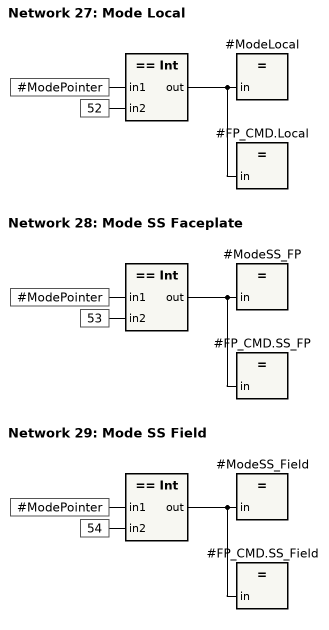
   #ModeLocal := #ModePointer = 52;
   #FP_CMD.Local := #ModeLocal;
END_REGION

REGION Network 28: Mode SS Faceplate
   #ModeSS_FP := #ModePointer = 53;
   #FP_CMD.SS_FP := #ModeSS_FP;
END_REGION

REGION Network 29: Mode SS Field
   #ModeSS_Field := #ModePointer = 54;
   #FP_CMD.SS_Field := #ModeSS_Field;
END_REGION

REGION Network 30: FACEPLATE COMMANDS (Pulse Type)
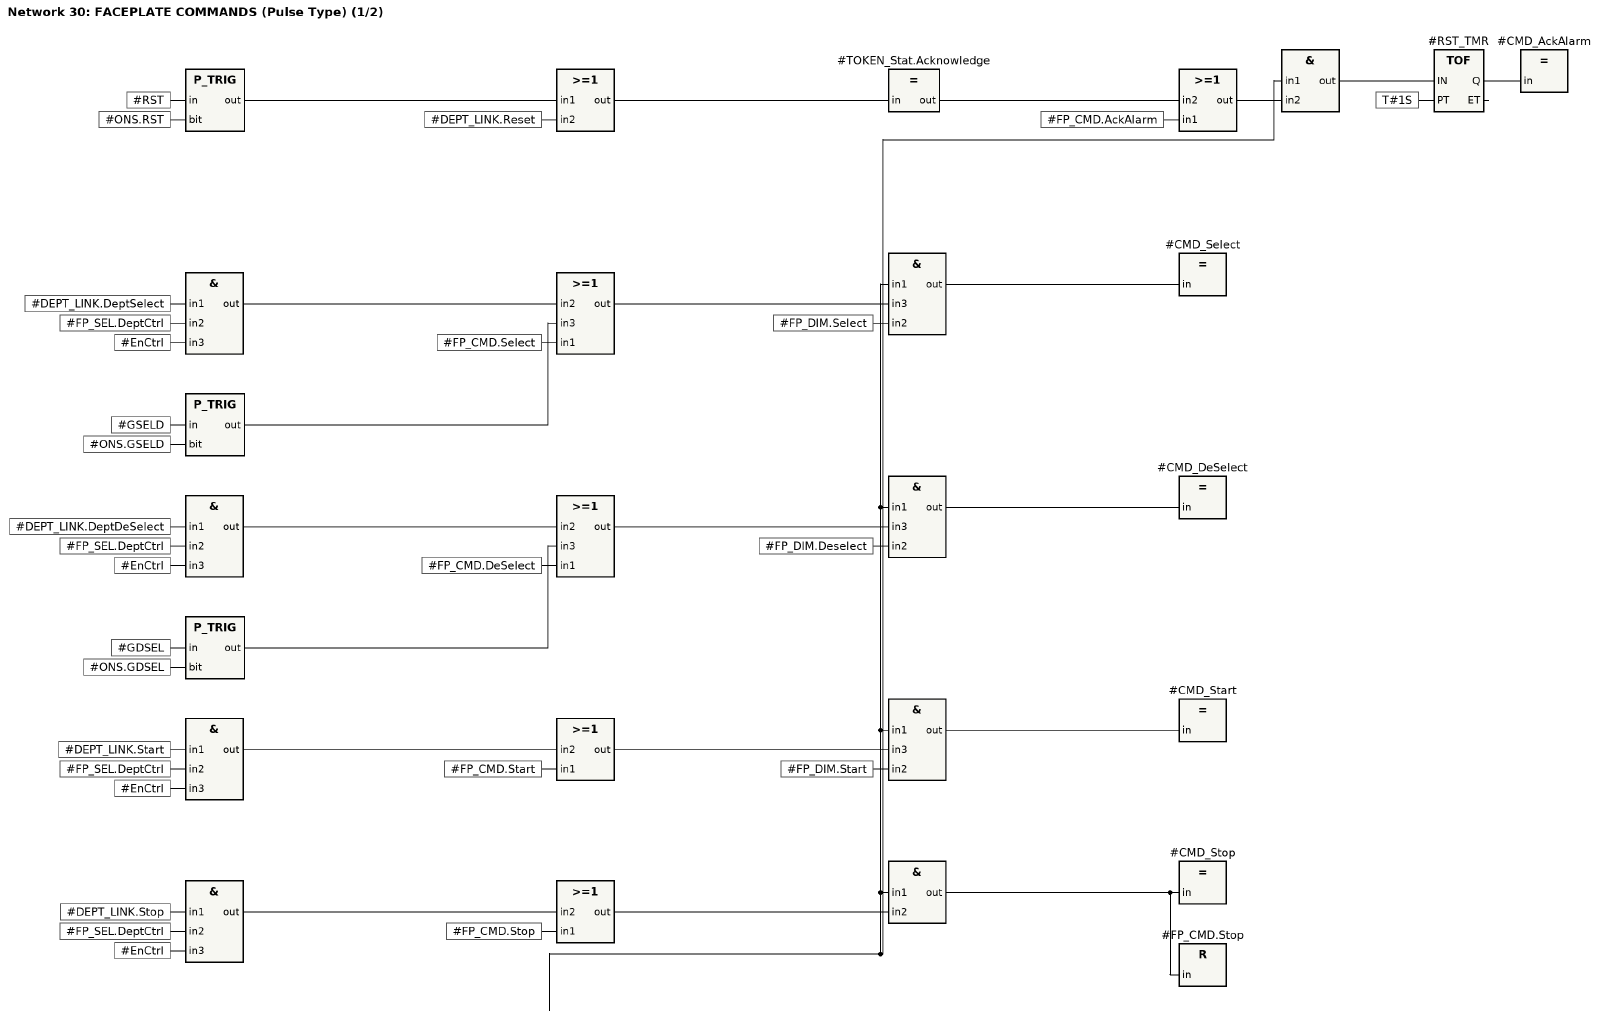
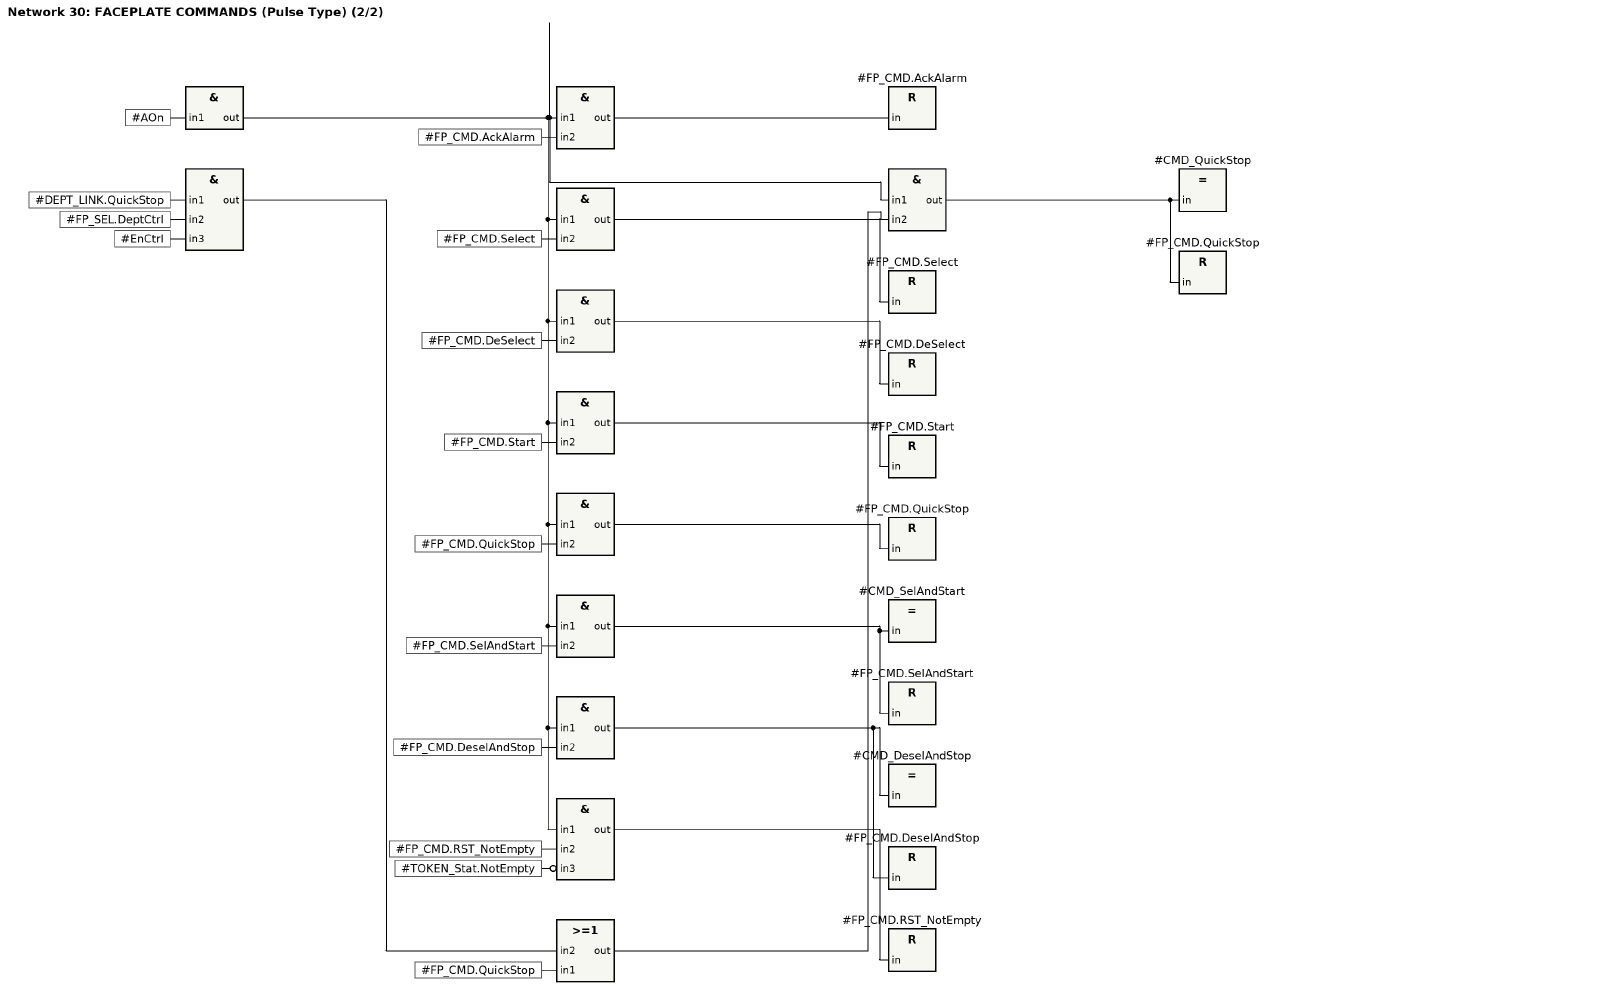
   #_w1 := #RST AND NOT #ONS.RST;   // rising edge
   #ONS.RST := #RST;
   #TOKEN_Stat.Acknowledge := #_w1 OR #DEPT_LINK.Reset;
   #RST_TMR(IN := #AOn AND (#TOKEN_Stat.Acknowledge OR #FP_CMD.AckAlarm), PT := T#1S);   // TOF
   #CMD_AckAlarm := #RST_TMR.Q;
   IF #AOn AND #FP_CMD.AckAlarm THEN #FP_CMD.AckAlarm := FALSE; END_IF;
   #_w2 := #GSELD AND NOT #ONS.GSELD;   // rising edge
   #ONS.GSELD := #GSELD;
   #CMD_Select := #AOn AND ((#DEPT_LINK.DeptSelect AND #FP_SEL.DeptCtrl AND #EnCtrl) OR #_w2 OR #FP_CMD.Select) AND #FP_DIM.Select;
   IF #AOn AND #FP_CMD.Select THEN #FP_CMD.Select := FALSE; END_IF;
   #_w3 := #GDSEL AND NOT #ONS.GDSEL;   // rising edge
   #ONS.GDSEL := #GDSEL;
   #CMD_DeSelect := #AOn AND ((#DEPT_LINK.DeptDeSelect AND #FP_SEL.DeptCtrl AND #EnCtrl) OR #_w3 OR #FP_CMD.DeSelect) AND #FP_DIM.Deselect;
   IF #AOn AND #FP_CMD.DeSelect THEN #FP_CMD.DeSelect := FALSE; END_IF;
   #CMD_Start := #AOn AND ((#DEPT_LINK.Start AND #FP_SEL.DeptCtrl AND #EnCtrl) OR #FP_CMD.Start) AND #FP_DIM.Start;
   IF #AOn AND #FP_CMD.Start THEN #FP_CMD.Start := FALSE; END_IF;
   #CMD_Stop := #AOn AND ((#DEPT_LINK.Stop AND #FP_SEL.DeptCtrl AND #EnCtrl) OR #FP_CMD.Stop);
   IF #CMD_Stop THEN #FP_CMD.Stop := FALSE; END_IF;
   #CMD_QuickStop := #AOn AND ((#DEPT_LINK.QuickStop AND #FP_SEL.DeptCtrl AND #EnCtrl) OR #FP_CMD.QuickStop);
   IF #CMD_QuickStop THEN #FP_CMD.QuickStop := FALSE; END_IF;
   IF #AOn AND #FP_CMD.QuickStop THEN #FP_CMD.QuickStop := FALSE; END_IF;
   #CMD_SelAndStart := #AOn AND #FP_CMD.SelAndStart;
   IF #CMD_SelAndStart THEN #FP_CMD.SelAndStart := FALSE; END_IF;
   #CMD_DeselAndStop := #AOn AND #FP_CMD.DeselAndStop;
   IF #CMD_DeselAndStop THEN #FP_CMD.DeselAndStop := FALSE; END_IF;
   IF #AOn AND #FP_CMD.RST_NotEmpty AND NOT #TOKEN_Stat.NotEmpty THEN #FP_CMD.RST_NotEmpty := FALSE; END_IF;
END_REGION

REGION Network 31: Start Warning timer
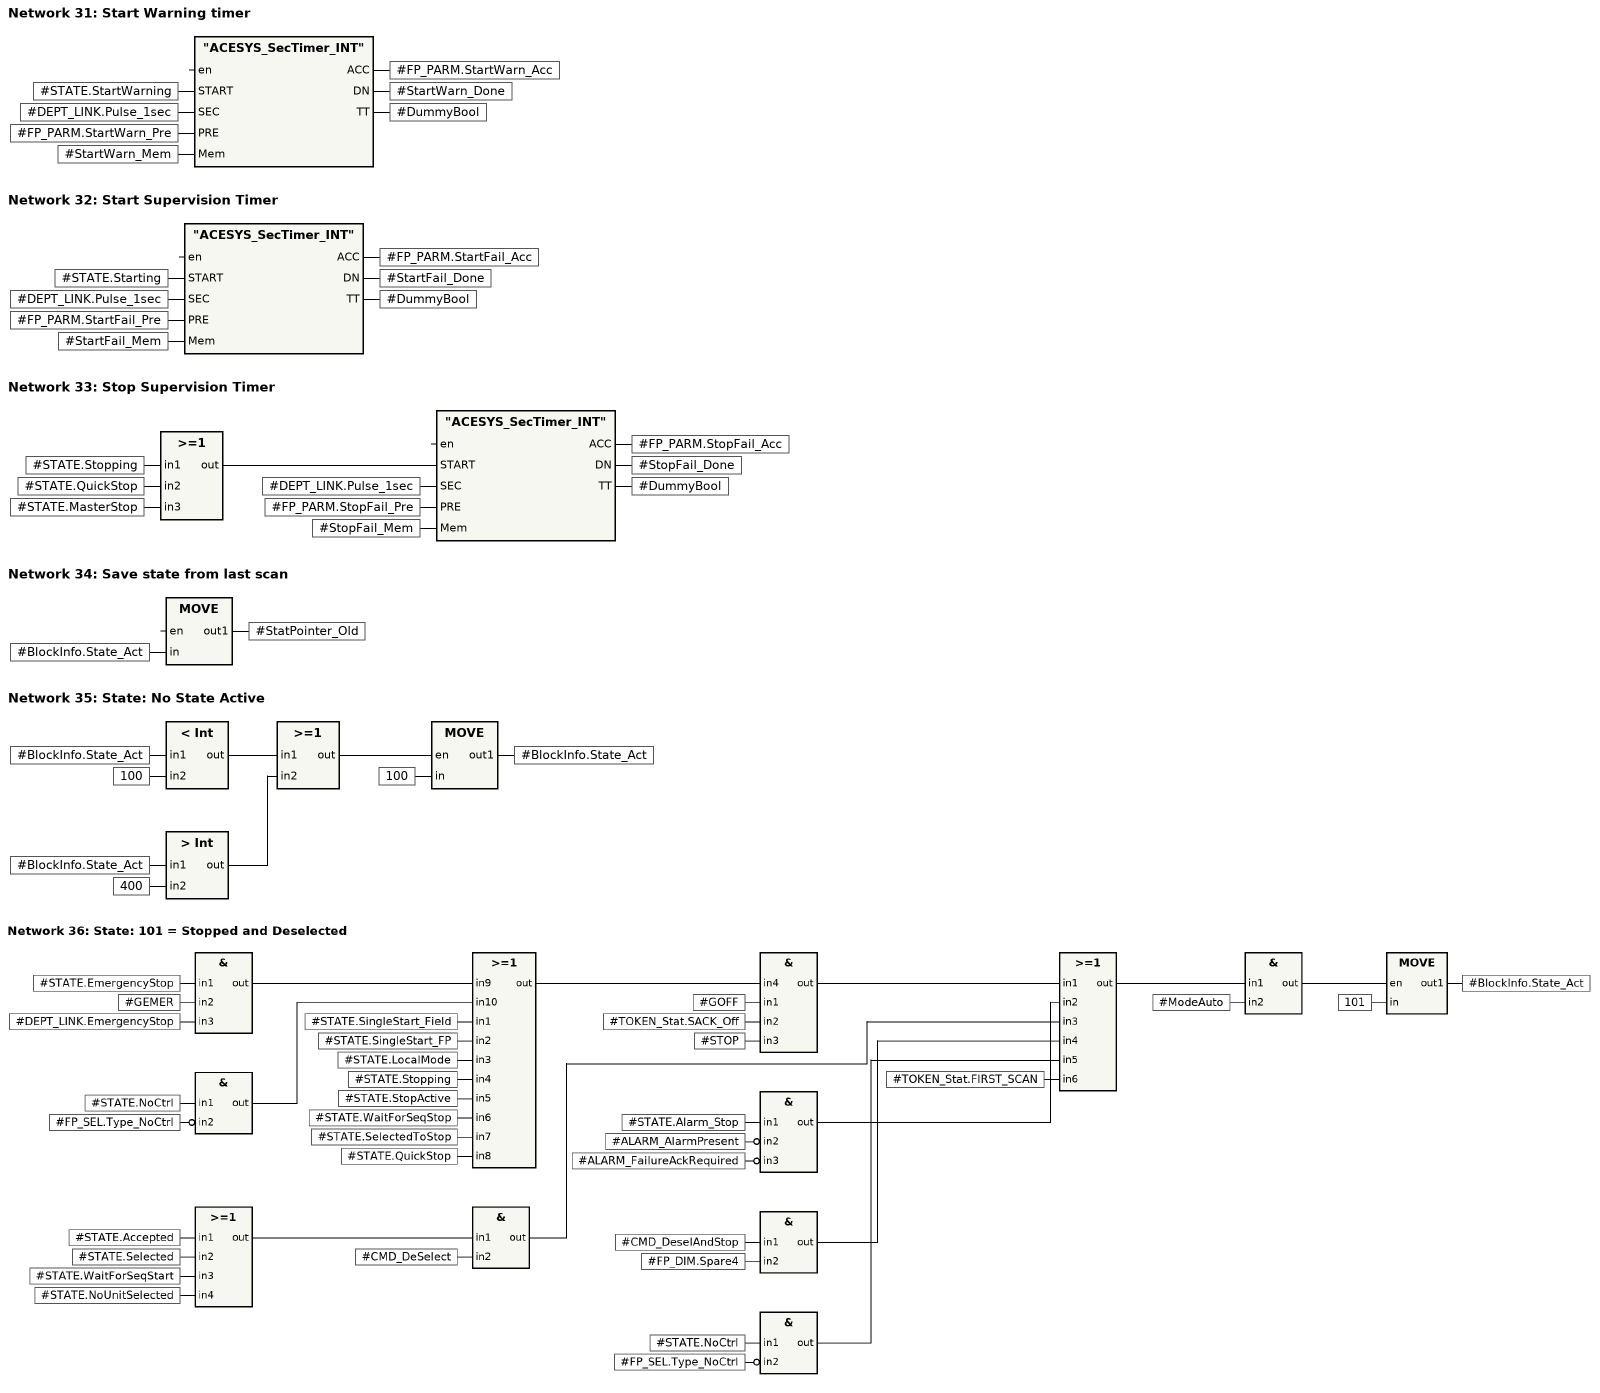
   "ACESYS_SecTimer_INT"(START := #STATE.StartWarning,
                         SEC := #DEPT_LINK.Pulse_1sec,
                         PRE := #FP_PARM.StartWarn_Pre,
                         Mem := #StartWarn_Mem,
                         ACC => #FP_PARM.StartWarn_Acc,
                         DN => #StartWarn_Done,
                         TT => #DummyBool);
END_REGION

REGION Network 32: Start Supervision Timer
   "ACESYS_SecTimer_INT"(START := #STATE.Starting,
                         SEC := #DEPT_LINK.Pulse_1sec,
                         PRE := #FP_PARM.StartFail_Pre,
                         Mem := #StartFail_Mem,
                         ACC => #FP_PARM.StartFail_Acc,
                         DN => #StartFail_Done,
                         TT => #DummyBool);
END_REGION

REGION Network 33: Stop Supervision Timer
   "ACESYS_SecTimer_INT"(START := #STATE.Stopping OR #STATE.QuickStop OR #STATE.MasterStop,
                         SEC := #DEPT_LINK.Pulse_1sec,
                         PRE := #FP_PARM.StopFail_Pre,
                         Mem := #StopFail_Mem,
                         ACC => #FP_PARM.StopFail_Acc,
                         DN => #StopFail_Done,
                         TT => #DummyBool);
END_REGION

REGION Network 34: Save state from last scan
   #StatPointer_Old := #BlockInfo.State_Act;
END_REGION

REGION Network 35: State: No State Active
   IF (#BlockInfo.State_Act < 100) OR (#BlockInfo.State_Act > 400) THEN #BlockInfo.State_Act := 100; END_IF;
END_REGION

REGION Network 36: State: 101 = Stopped and Deselected
   // Build 004 - 05.Aug.2021 (MIA-US): Transition from State_WaitForSeqStop added
   IF ((((#STATE.EmergencyStop AND #GEMER AND #DEPT_LINK.EmergencyStop) OR (#STATE.NoCtrl AND NOT #FP_SEL.Type_NoCtrl) OR #STATE.SingleStart_Field OR #STATE.SingleStart_FP OR #STATE.LocalMode OR #STATE.Stopping OR #STATE.StopActive OR #STATE.WaitForSeqStop OR #STATE.SelectedToStop OR #STATE.QuickStop) AND #GOFF AND #TOKEN_Stat.SACK_Off AND #STOP) OR (#STATE.Alarm_Stop AND NOT #ALARM_AlarmPresent AND NOT #ALARM_FailureAckRequired) OR ((#STATE.Accepted OR #STATE.Selected OR #STATE.WaitForSeqStart OR #STATE.NoUnitSelected) AND #CMD_DeSelect) OR (#CMD_DeselAndStop AND #FP_DIM.Spare4) OR (#STATE.NoCtrl AND NOT #FP_SEL.Type_NoCtrl) OR #TOKEN_Stat.FIRST_SCAN) AND #ModeAuto THEN
       #BlockInfo.State_Act := 101;
   END_IF;
END_REGION

REGION Network 37 (SCL): Transfer Interlock OK to Stat
   #OUT.INTL_OK_STAT := PEEK_BOOL(area :=16#84, dbNumber := #BlockInfo.DB_Number, byteOffset := 2, bitOffset := 0);
   #OUT.INTL_SEQ_STR_OK_STAT := PEEK_BOOL(area := 16#84, dbNumber := #BlockInfo.DB_Number, byteOffset := 4, bitOffset := 0);
   #OUT.INTL_SEQ_STP_OK_STAT := PEEK_BOOL(area := 16#84, dbNumber := #BlockInfo.DB_Number, byteOffset := 6, bitOffset := 0);
END_REGION

REGION Network 38: Conditions for Accept
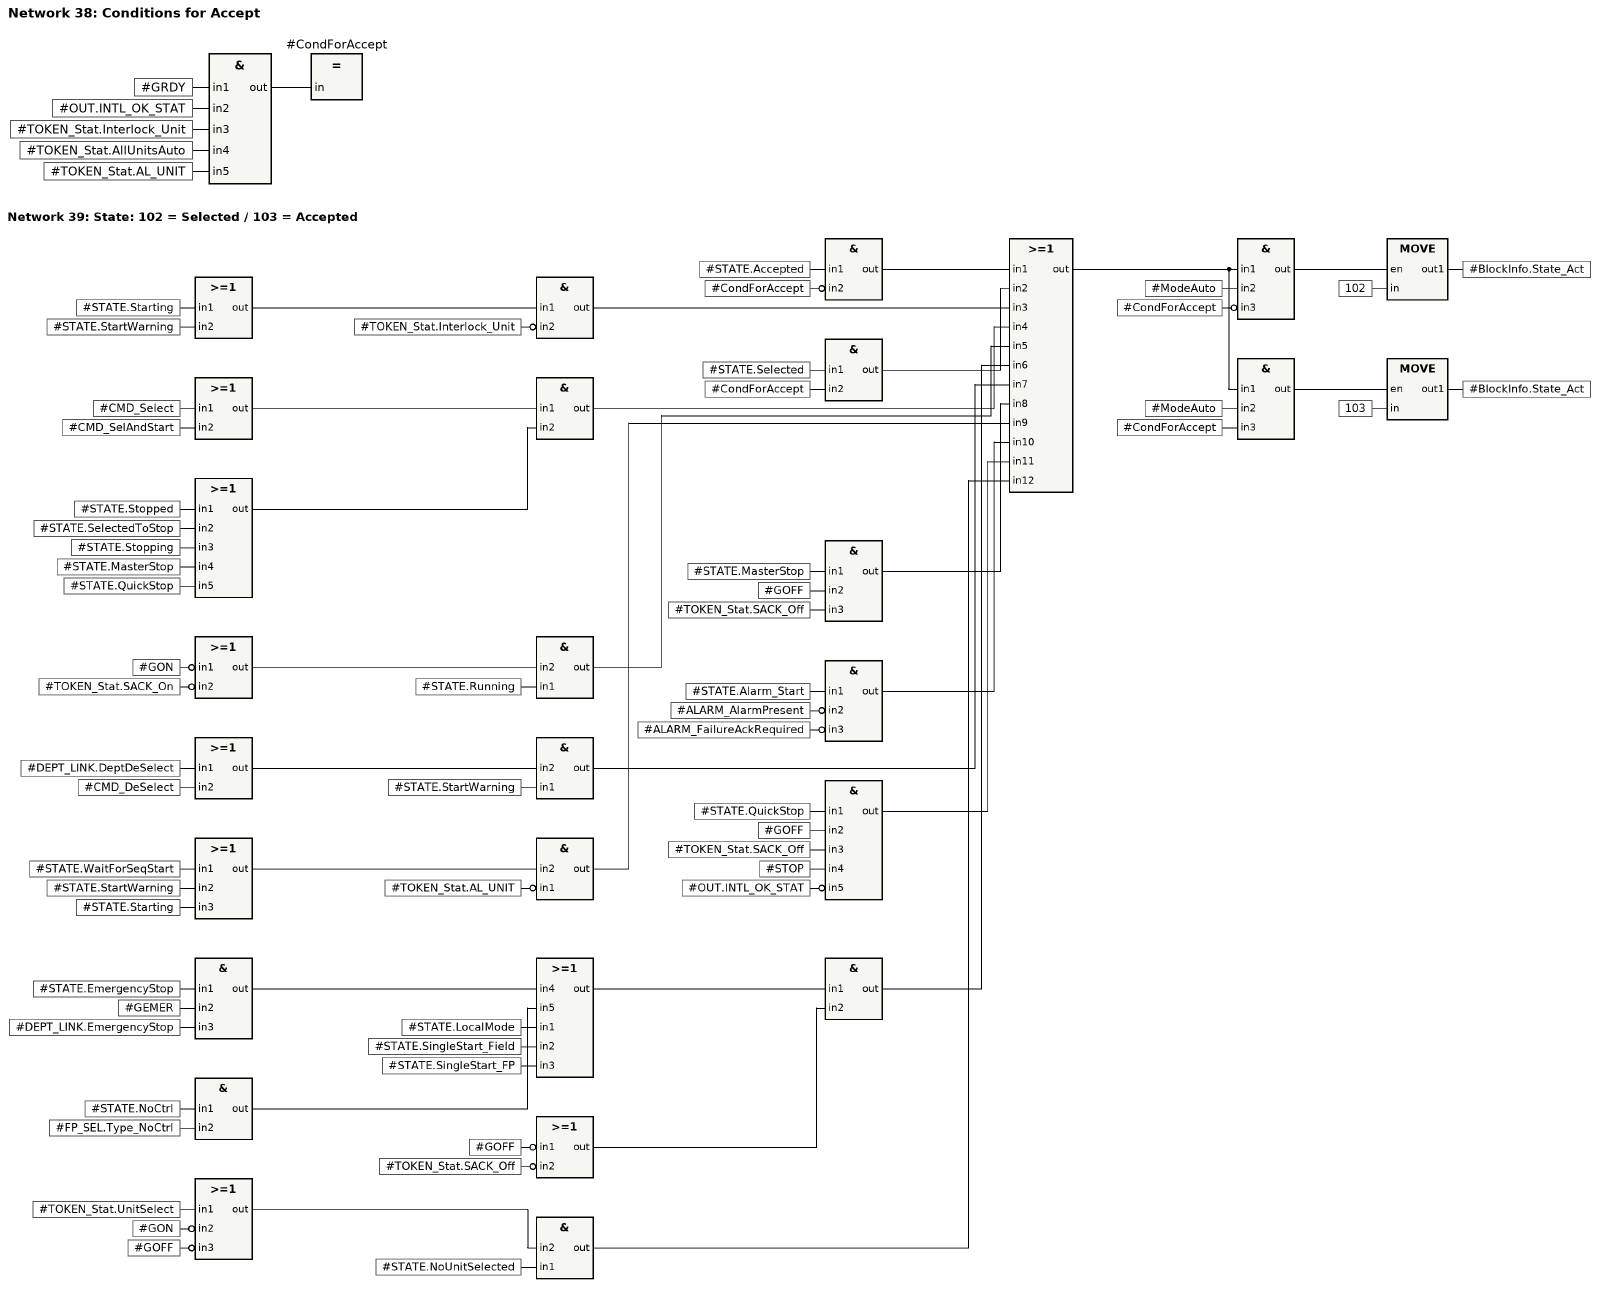
   #CondForAccept := #GRDY AND #OUT.INTL_OK_STAT AND #TOKEN_Stat.Interlock_Unit AND #TOKEN_Stat.AllUnitsAuto AND #TOKEN_Stat.AL_UNIT;
END_REGION

REGION Network 39: State: 102 = Selected / 103 = Accepted
   #_w1 := (#STATE.Accepted AND NOT #CondForAccept) OR (#STATE.Selected AND #CondForAccept) OR ((#STATE.Starting OR #STATE.StartWarning) AND NOT #TOKEN_Stat.Interlock_Unit) OR ((#CMD_Select OR #CMD_SelAndStart) AND (#STATE.Stopped OR #STATE.SelectedToStop OR #STATE.Stopping OR #STATE.MasterStop OR #STATE.QuickStop)) OR ((NOT #GON OR NOT #TOKEN_Stat.SACK_On) AND #STATE.Running) OR (((#STATE.EmergencyStop AND #GEMER AND #DEPT_LINK.EmergencyStop) OR (#STATE.NoCtrl AND #FP_SEL.Type_NoCtrl) OR #STATE.LocalMode OR #STATE.SingleStart_Field OR #STATE.SingleStart_FP) AND (NOT #GOFF OR NOT #TOKEN_Stat.SACK_Off)) OR ((#DEPT_LINK.DeptDeSelect OR #CMD_DeSelect) AND #STATE.StartWarning) OR (#STATE.MasterStop AND #GOFF AND #TOKEN_Stat.SACK_Off) OR ((#STATE.WaitForSeqStart OR #STATE.StartWarning OR #STATE.Starting) AND NOT #TOKEN_Stat.AL_UNIT) OR (#STATE.Alarm_Start AND NOT #ALARM_AlarmPresent AND NOT #ALARM_FailureAckRequired) OR (#STATE.QuickStop AND #GOFF AND #TOKEN_Stat.SACK_Off AND #STOP AND NOT #OUT.INTL_OK_STAT) OR ((#TOKEN_Stat.UnitSelect OR NOT #GON OR NOT #GOFF) AND #STATE.NoUnitSelected);
   IF #_w1 AND #ModeAuto AND NOT #CondForAccept THEN #BlockInfo.State_Act := 102; END_IF;
   IF #_w1 AND #ModeAuto AND #CondForAccept THEN #BlockInfo.State_Act := 103; END_IF;
END_REGION

REGION Network 40: State: 104 = Wait for Sequence Start
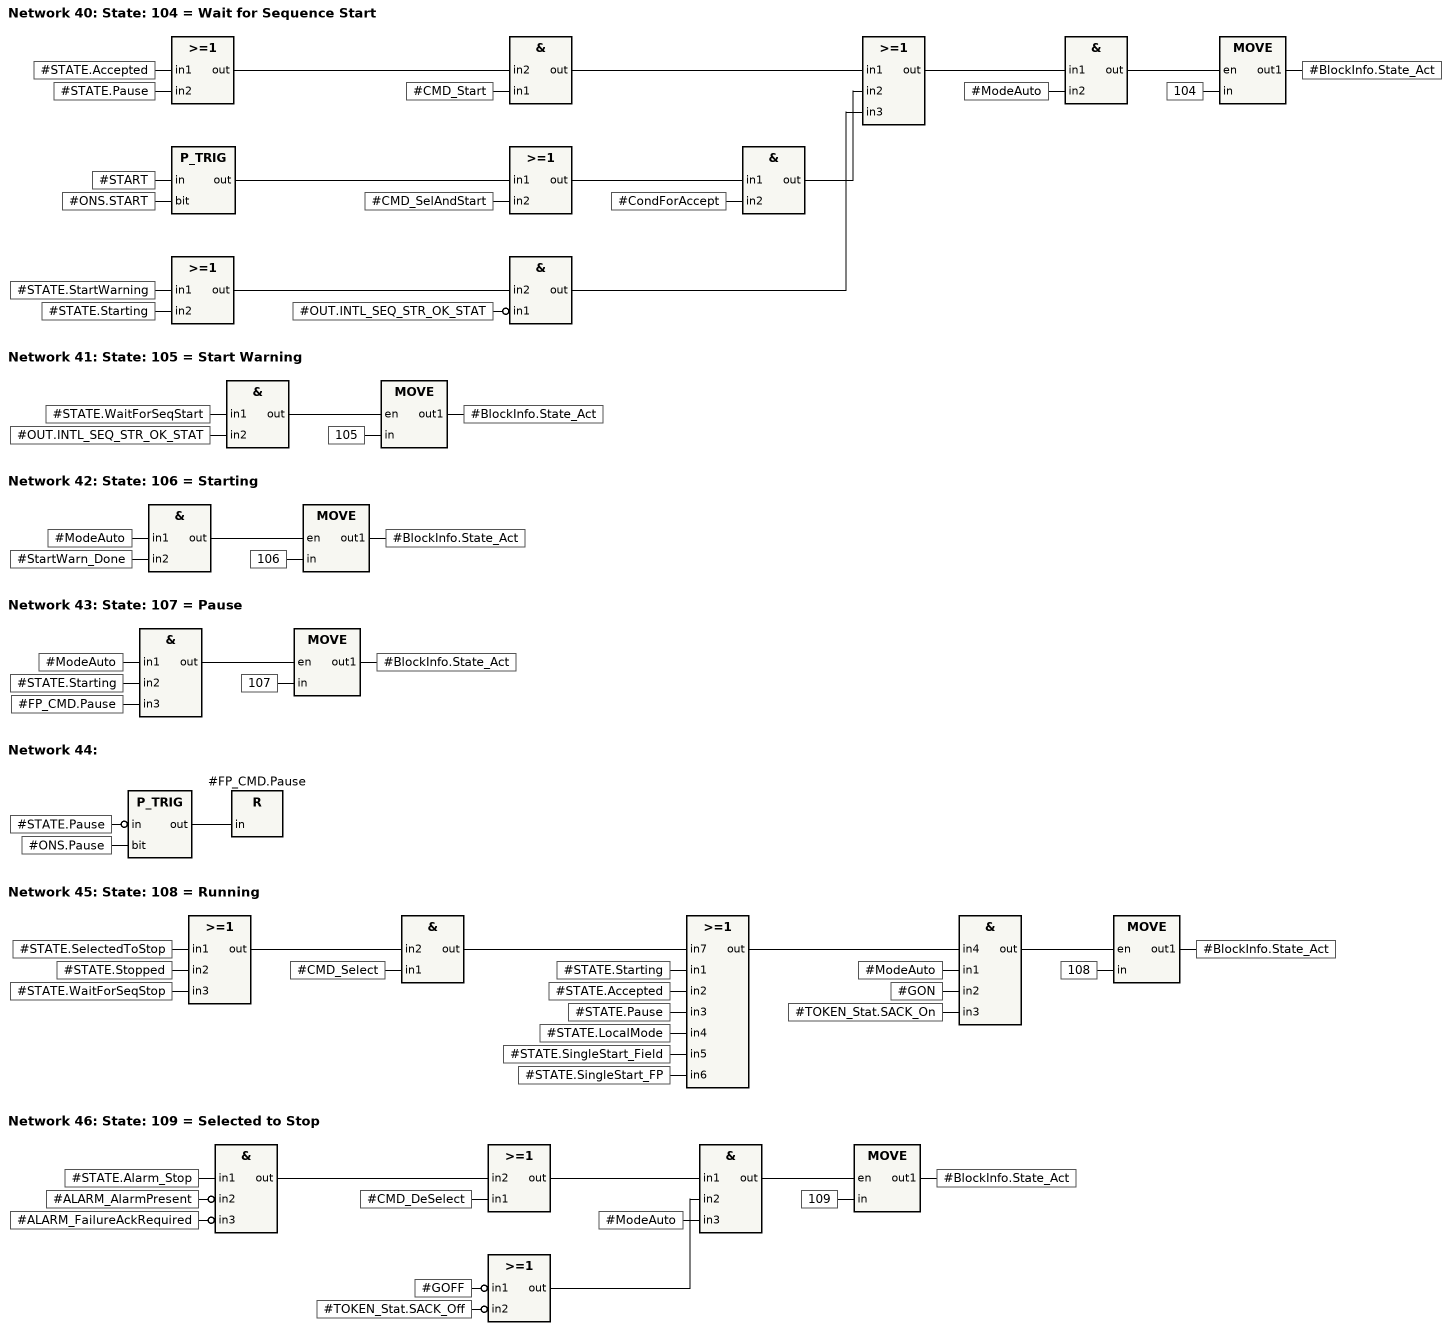
   #_w1 := #START AND NOT #ONS.START;   // rising edge
   #ONS.START := #START;
   IF (((#STATE.Accepted OR #STATE.Pause) AND #CMD_Start) OR ((#_w1 OR #CMD_SelAndStart) AND #CondForAccept) OR ((#STATE.StartWarning OR #STATE.Starting) AND NOT #OUT.INTL_SEQ_STR_OK_STAT)) AND #ModeAuto THEN
       #BlockInfo.State_Act := 104;
   END_IF;
END_REGION

REGION Network 41: State: 105 = Start Warning
   IF #STATE.WaitForSeqStart AND #OUT.INTL_SEQ_STR_OK_STAT THEN #BlockInfo.State_Act := 105; END_IF;
END_REGION

REGION Network 42: State: 106 = Starting
   IF #ModeAuto AND #StartWarn_Done THEN #BlockInfo.State_Act := 106; END_IF;
END_REGION

REGION Network 43: State: 107 = Pause
   IF #ModeAuto AND #STATE.Starting AND #FP_CMD.Pause THEN #BlockInfo.State_Act := 107; END_IF;
END_REGION

REGION Network 44
   #_w1 := NOT #STATE.Pause AND NOT #ONS.Pause;   // rising edge
   #ONS.Pause := NOT #STATE.Pause;
   IF #_w1 THEN #FP_CMD.Pause := FALSE; END_IF;
END_REGION

REGION Network 45: State: 108 = Running
   IF (((#STATE.SelectedToStop OR #STATE.Stopped OR #STATE.WaitForSeqStop) AND #CMD_Select) OR #STATE.Starting OR #STATE.Accepted OR #STATE.Pause OR #STATE.LocalMode OR #STATE.SingleStart_Field OR #STATE.SingleStart_FP) AND #ModeAuto AND #GON AND #TOKEN_Stat.SACK_On THEN
       #BlockInfo.State_Act := 108;
   END_IF;
END_REGION

REGION Network 46: State: 109 = Selected to Stop
   IF ((#STATE.Alarm_Stop AND NOT #ALARM_AlarmPresent AND NOT #ALARM_FailureAckRequired) OR #CMD_DeSelect) AND (NOT #GOFF OR NOT #TOKEN_Stat.SACK_Off) AND #ModeAuto THEN
       #BlockInfo.State_Act := 109;
   END_IF;
END_REGION

REGION Network 47: State: 110 = Wait for Sequence Stop
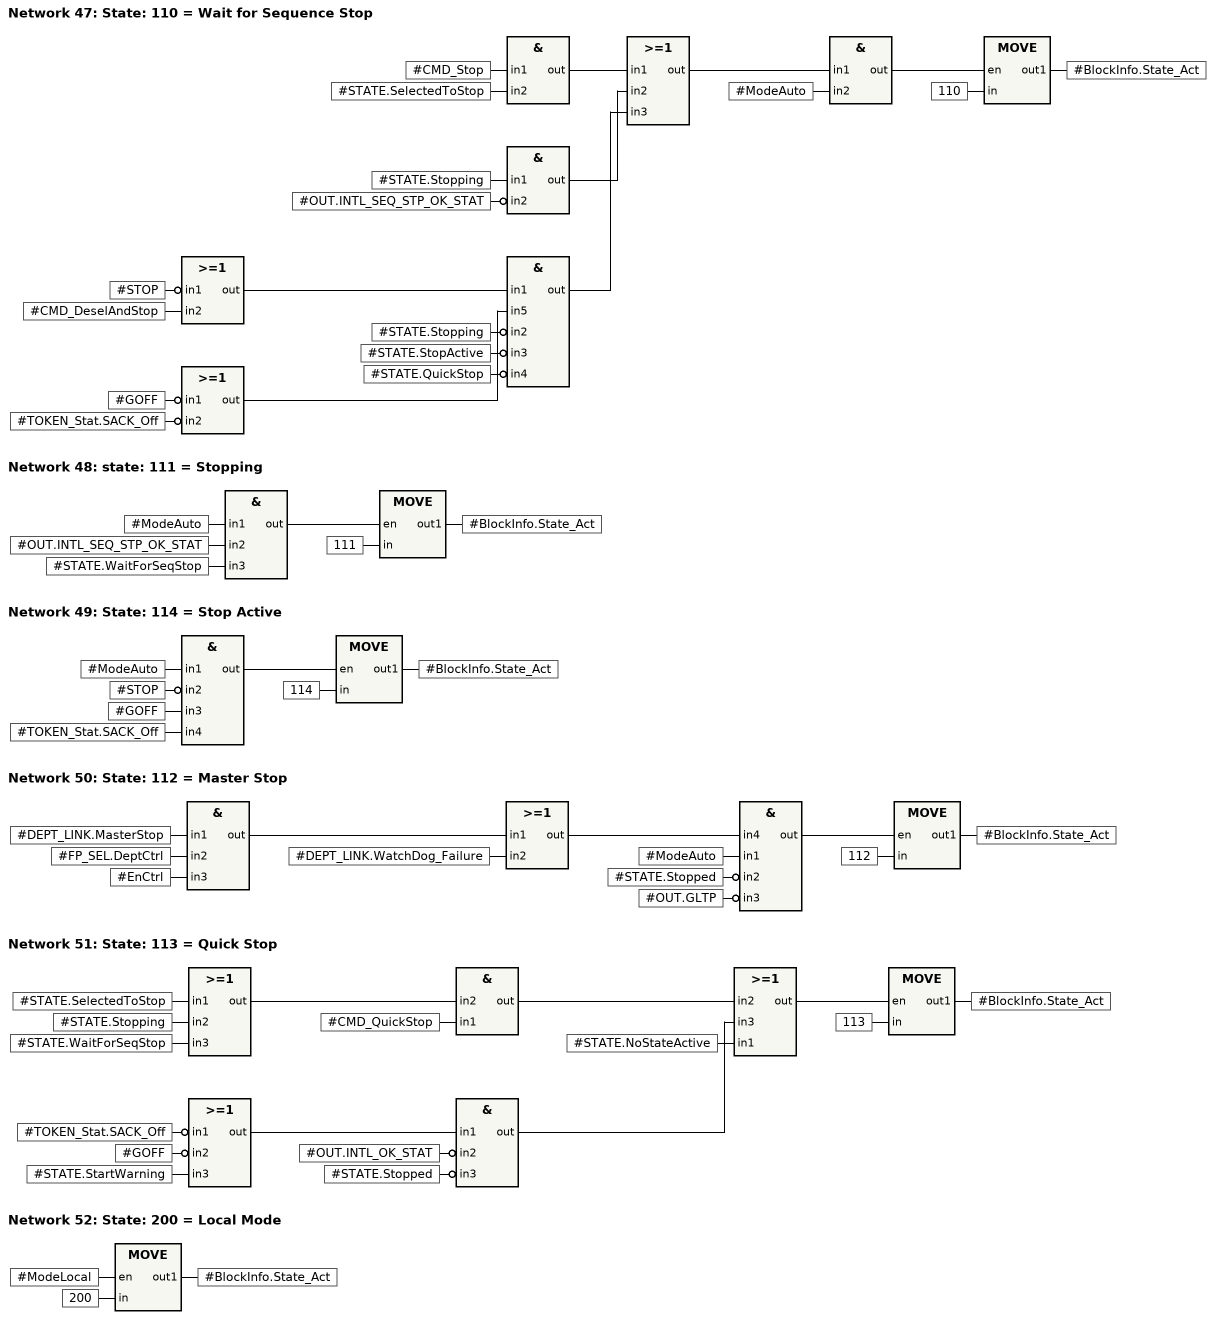
   IF ((#CMD_Stop AND #STATE.SelectedToStop) OR (#STATE.Stopping AND NOT #OUT.INTL_SEQ_STP_OK_STAT) OR ((NOT #STOP OR #CMD_DeselAndStop) AND (NOT #GOFF OR NOT #TOKEN_Stat.SACK_Off) AND NOT #STATE.Stopping AND NOT #STATE.StopActive AND NOT #STATE.QuickStop)) AND #ModeAuto THEN
       #BlockInfo.State_Act := 110;
   END_IF;
END_REGION

REGION Network 48: state: 111 = Stopping
   IF #ModeAuto AND #OUT.INTL_SEQ_STP_OK_STAT AND #STATE.WaitForSeqStop THEN
       #BlockInfo.State_Act := 111;
   END_IF;
END_REGION

REGION Network 49: State: 114 = Stop Active
   IF #ModeAuto AND NOT #STOP AND #GOFF AND #TOKEN_Stat.SACK_Off THEN #BlockInfo.State_Act := 114; END_IF;
END_REGION

REGION Network 50: State: 112 = Master Stop
   IF ((#DEPT_LINK.MasterStop AND #FP_SEL.DeptCtrl AND #EnCtrl) OR #DEPT_LINK.WatchDog_Failure) AND #ModeAuto AND NOT #STATE.Stopped AND NOT #OUT.GLTP THEN
       #BlockInfo.State_Act := 112;
   END_IF;
END_REGION

REGION Network 51: State: 113 = Quick Stop
   // Build 002 - 17.Dec.2019 (MIA-US): Added STATE.StartWarning to allow transition to "Interlock" state when INTL=0 during start warning
   // Build 003 - 24.Jun.2020 (MIA-US): Removed TOKEN_Stat.SACK_On
   IF ((#STATE.SelectedToStop OR #STATE.Stopping OR #STATE.WaitForSeqStop) AND #CMD_QuickStop) OR ((NOT #TOKEN_Stat.SACK_Off OR NOT #GOFF OR #STATE.StartWarning) AND NOT #OUT.INTL_OK_STAT AND NOT #STATE.Stopped) OR #STATE.NoStateActive THEN
       #BlockInfo.State_Act := 113;
   END_IF;
END_REGION

REGION Network 52: State: 200 = Local Mode
   IF #ModeLocal THEN #BlockInfo.State_Act := 200; END_IF;
END_REGION

REGION Network 53: State: 250 = Single Start from Faceplate
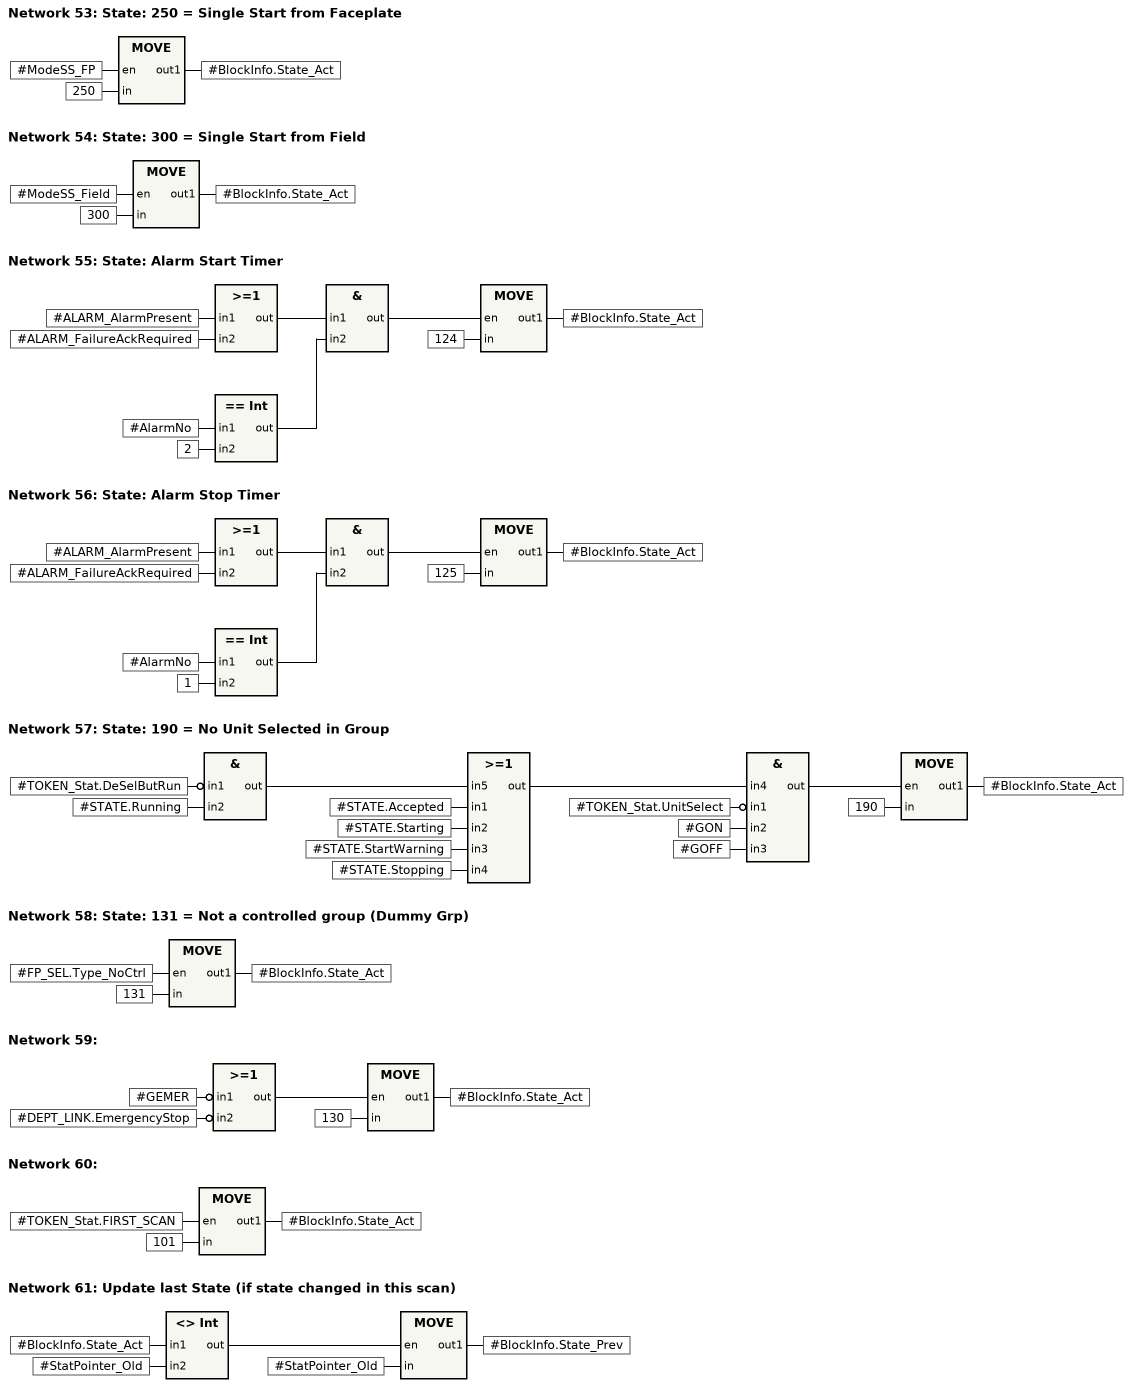
   IF #ModeSS_FP THEN #BlockInfo.State_Act := 250; END_IF;
END_REGION

REGION Network 54: State: 300 = Single Start from Field
   IF #ModeSS_Field THEN #BlockInfo.State_Act := 300; END_IF;
END_REGION

REGION Network 55: State: Alarm Start Timer
   IF (#ALARM_AlarmPresent OR #ALARM_FailureAckRequired) AND (#AlarmNo = 2) THEN
       #BlockInfo.State_Act := 124;
   END_IF;
END_REGION

REGION Network 56: State: Alarm Stop Timer
   IF (#ALARM_AlarmPresent OR #ALARM_FailureAckRequired) AND (#AlarmNo = 1) THEN
       #BlockInfo.State_Act := 125;
   END_IF;
END_REGION

REGION Network 57: State: 190 = No Unit Selected in Group
   IF ((NOT #TOKEN_Stat.DeSelButRun AND #STATE.Running) OR #STATE.Accepted OR #STATE.Starting OR #STATE.StartWarning OR #STATE.Stopping) AND NOT #TOKEN_Stat.UnitSelect AND #GON AND #GOFF THEN
       #BlockInfo.State_Act := 190;
   END_IF;
END_REGION

REGION Network 58: State: 131 = Not a controlled group (Dummy Grp)
   IF #FP_SEL.Type_NoCtrl THEN #BlockInfo.State_Act := 131; END_IF;
END_REGION

REGION Network 59
   IF NOT #GEMER OR NOT #DEPT_LINK.EmergencyStop THEN #BlockInfo.State_Act := 130; END_IF;
END_REGION

REGION Network 60
   IF #TOKEN_Stat.FIRST_SCAN THEN #BlockInfo.State_Act := 101; END_IF;
END_REGION

REGION Network 61: Update last State (if state changed in this scan)
   IF #BlockInfo.State_Act <> #StatPointer_Old THEN #BlockInfo.State_Prev := #StatPointer_Old; END_IF;
END_REGION

REGION Network 62: State Status Flag - No Unit Selected
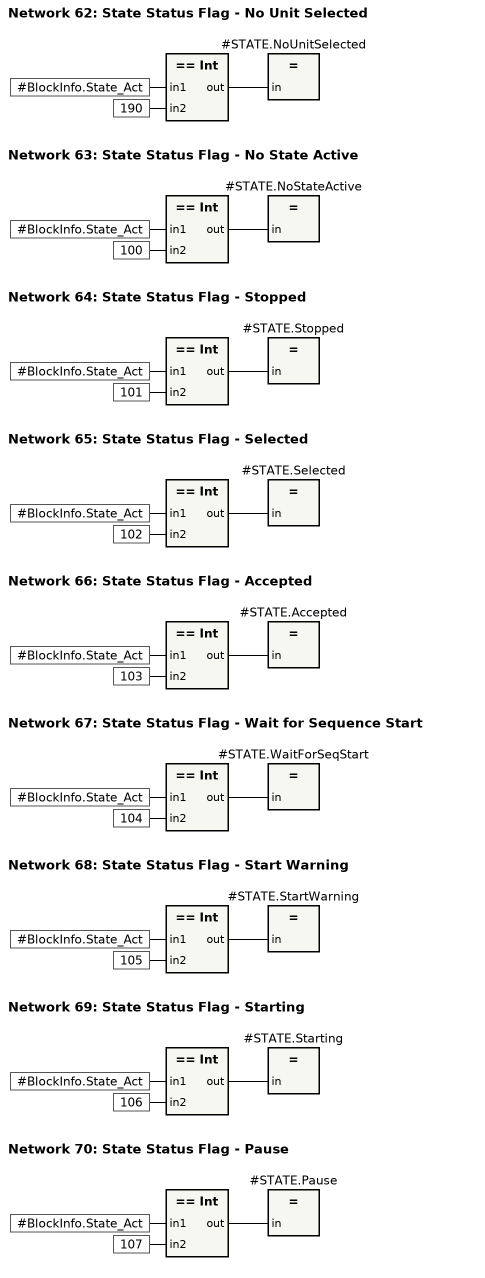
   #STATE.NoUnitSelected := #BlockInfo.State_Act = 190;
END_REGION

REGION Network 63: State Status Flag - No State Active
   #STATE.NoStateActive := #BlockInfo.State_Act = 100;
END_REGION

REGION Network 64: State Status Flag - Stopped
   #STATE.Stopped := #BlockInfo.State_Act = 101;
END_REGION

REGION Network 65: State Status Flag - Selected
   #STATE.Selected := #BlockInfo.State_Act = 102;
END_REGION

REGION Network 66: State Status Flag - Accepted
   #STATE.Accepted := #BlockInfo.State_Act = 103;
END_REGION

REGION Network 67: State Status Flag - Wait for Sequence Start
   #STATE.WaitForSeqStart := #BlockInfo.State_Act = 104;
END_REGION

REGION Network 68: State Status Flag - Start Warning
   #STATE.StartWarning := #BlockInfo.State_Act = 105;
END_REGION

REGION Network 69: State Status Flag - Starting
   #STATE.Starting := #BlockInfo.State_Act = 106;
END_REGION

REGION Network 70: State Status Flag - Pause
   #STATE.Pause := #BlockInfo.State_Act = 107;
END_REGION

REGION Network 71: State Status Flag - Running
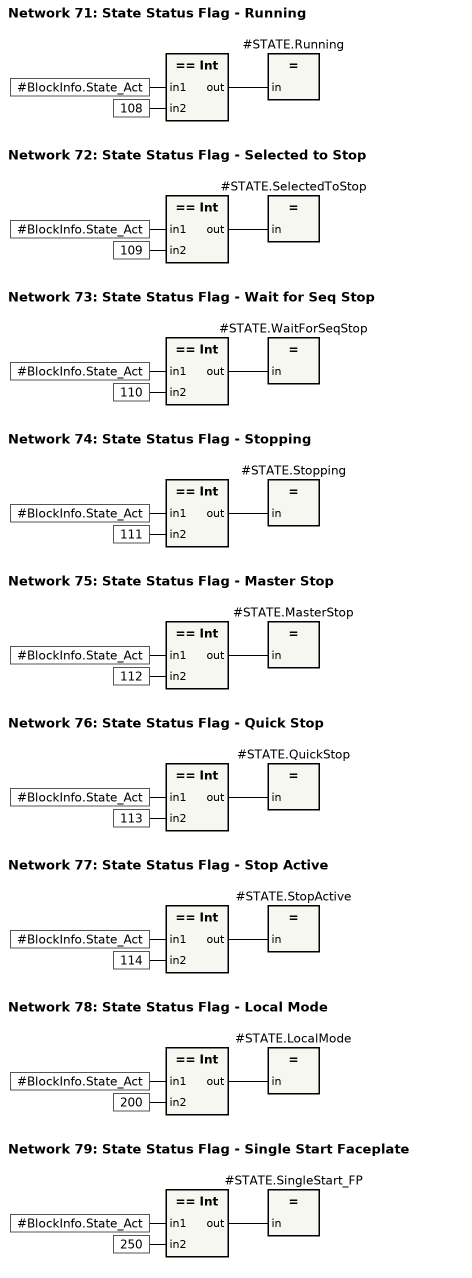
   #STATE.Running := #BlockInfo.State_Act = 108;
END_REGION

REGION Network 72: State Status Flag - Selected to Stop
   #STATE.SelectedToStop := #BlockInfo.State_Act = 109;
END_REGION

REGION Network 73: State Status Flag - Wait for Seq Stop
   #STATE.WaitForSeqStop := #BlockInfo.State_Act = 110;
END_REGION

REGION Network 74: State Status Flag - Stopping
   #STATE.Stopping := #BlockInfo.State_Act = 111;
END_REGION

REGION Network 75: State Status Flag - Master Stop
   #STATE.MasterStop := #BlockInfo.State_Act = 112;
END_REGION

REGION Network 76: State Status Flag - Quick Stop
   #STATE.QuickStop := #BlockInfo.State_Act = 113;
END_REGION

REGION Network 77: State Status Flag - Stop Active
   #STATE.StopActive := #BlockInfo.State_Act = 114;
END_REGION

REGION Network 78: State Status Flag - Local Mode
   #STATE.LocalMode := #BlockInfo.State_Act = 200;
END_REGION

REGION Network 79: State Status Flag - Single Start Faceplate
   #STATE.SingleStart_FP := #BlockInfo.State_Act = 250;
END_REGION

REGION Network 80: State Status Flag - Single Start Field
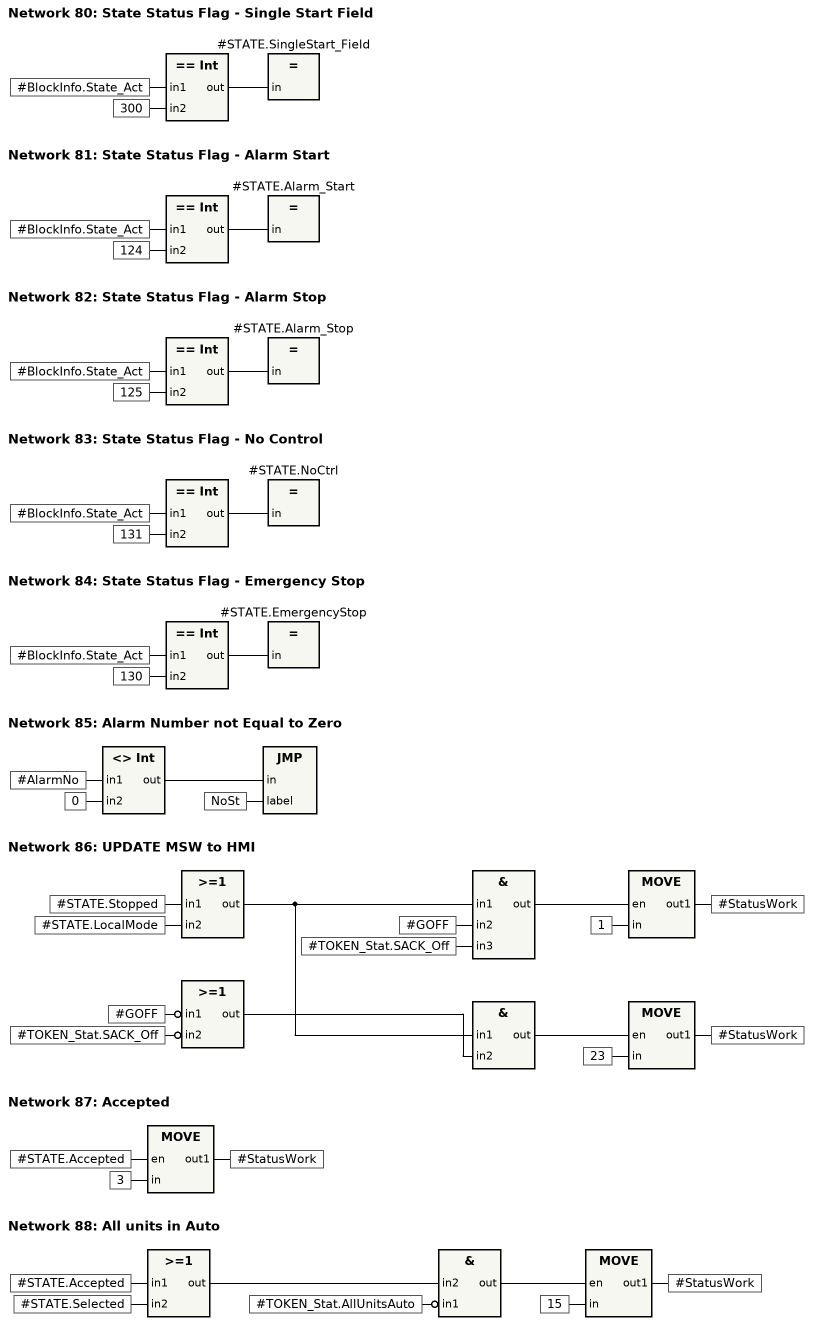
   #STATE.SingleStart_Field := #BlockInfo.State_Act = 300;
END_REGION

REGION Network 81: State Status Flag - Alarm Start
   #STATE.Alarm_Start := #BlockInfo.State_Act = 124;
END_REGION

REGION Network 82: State Status Flag - Alarm Stop
   #STATE.Alarm_Stop := #BlockInfo.State_Act = 125;
END_REGION

REGION Network 83: State Status Flag - No Control
   #STATE.NoCtrl := #BlockInfo.State_Act = 131;
END_REGION

REGION Network 84: State Status Flag - Emergency Stop
   #STATE.EmergencyStop := #BlockInfo.State_Act = 130;
END_REGION

REGION Network 85: Alarm Number not Equal to Zero
   IF #AlarmNo <> 0 THEN GOTO NoSt; END_IF;
END_REGION

REGION Network 86: UPDATE MSW to HMI
   // 1= Stopped, 23 = Ext. Started
   #_w1 := #STATE.Stopped OR #STATE.LocalMode;
   IF #_w1 AND #GOFF AND #TOKEN_Stat.SACK_Off THEN #StatusWork := 1; END_IF;
   IF #_w1 AND (NOT #GOFF OR NOT #TOKEN_Stat.SACK_Off) THEN #StatusWork := 23; END_IF;
END_REGION

REGION Network 87: Accepted
   IF #STATE.Accepted THEN #StatusWork := 3; END_IF;
END_REGION

REGION Network 88: All units in Auto
   IF (#STATE.Accepted OR #STATE.Selected) AND NOT #TOKEN_Stat.AllUnitsAuto THEN #StatusWork := 15; END_IF;
END_REGION

REGION Network 89: Start Warning
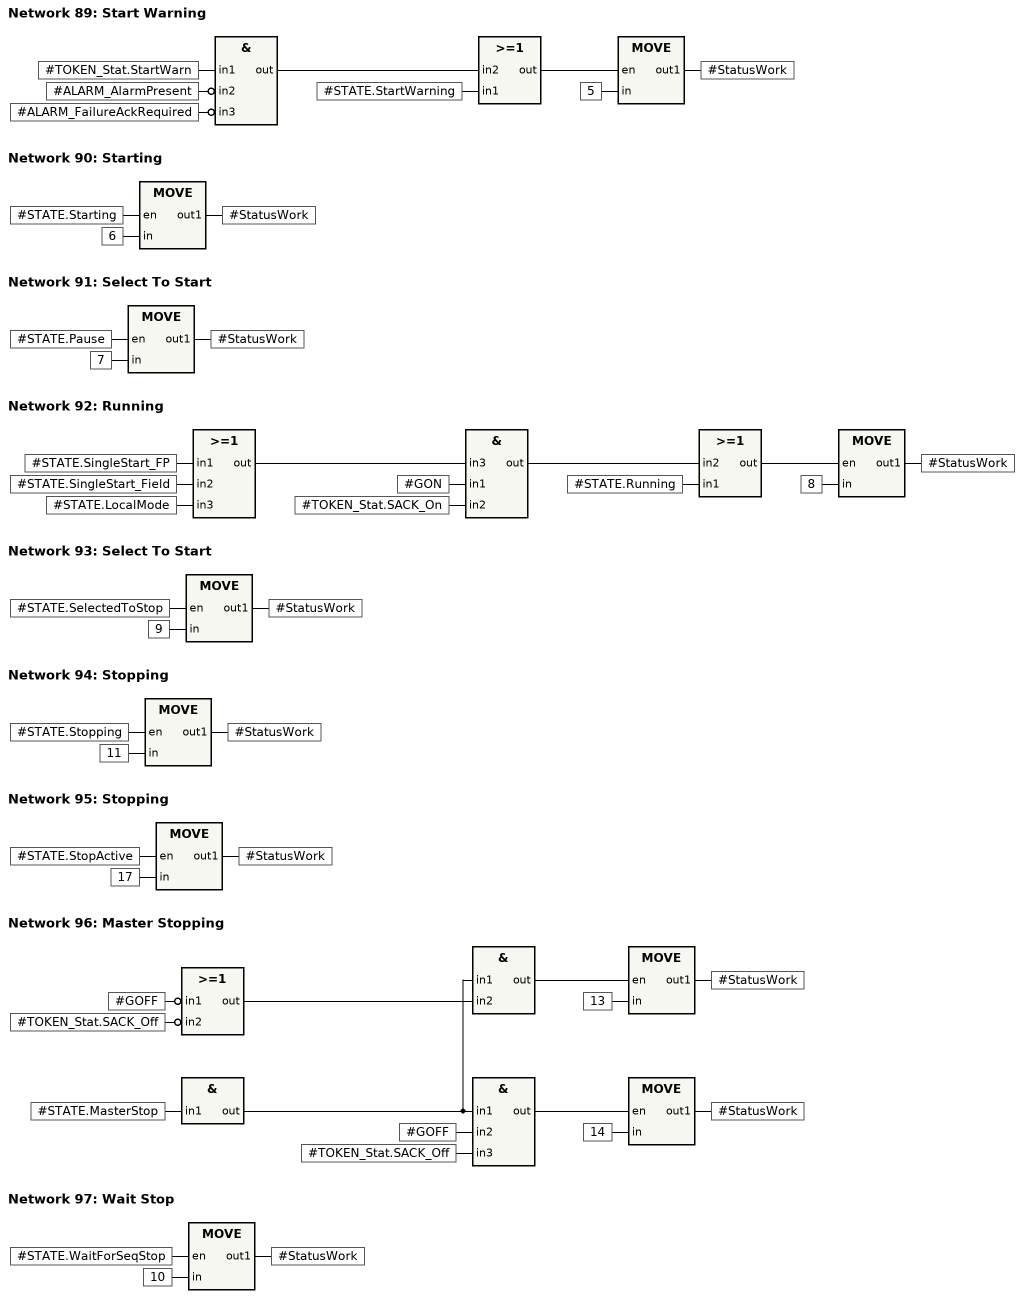
   IF (#TOKEN_Stat.StartWarn AND NOT #ALARM_AlarmPresent AND NOT #ALARM_FailureAckRequired) OR #STATE.StartWarning THEN
       #StatusWork := 5;
   END_IF;
END_REGION

REGION Network 90: Starting
   IF #STATE.Starting THEN #StatusWork := 6; END_IF;
END_REGION

REGION Network 91: Select To Start
   IF #STATE.Pause THEN #StatusWork := 7; END_IF;
END_REGION

REGION Network 92: Running
   IF ((#STATE.SingleStart_FP OR #STATE.SingleStart_Field OR #STATE.LocalMode) AND #GON AND #TOKEN_Stat.SACK_On) OR #STATE.Running THEN
       #StatusWork := 8;
   END_IF;
END_REGION

REGION Network 93: Select To Start
   IF #STATE.SelectedToStop THEN #StatusWork := 9; END_IF;
END_REGION

REGION Network 94: Stopping
   IF #STATE.Stopping THEN #StatusWork := 11; END_IF;
END_REGION

REGION Network 95: Stopping
   IF #STATE.StopActive THEN #StatusWork := 17; END_IF;
END_REGION

REGION Network 96: Master Stopping
   IF #STATE.MasterStop AND (NOT #GOFF OR NOT #TOKEN_Stat.SACK_Off) THEN #StatusWork := 13; END_IF;
   IF #STATE.MasterStop AND #GOFF AND #TOKEN_Stat.SACK_Off THEN #StatusWork := 14; END_IF;
END_REGION

REGION Network 97: Wait Stop
   IF #STATE.WaitForSeqStop THEN #StatusWork := 10; END_IF;
END_REGION

REGION Network 98: Wait Start
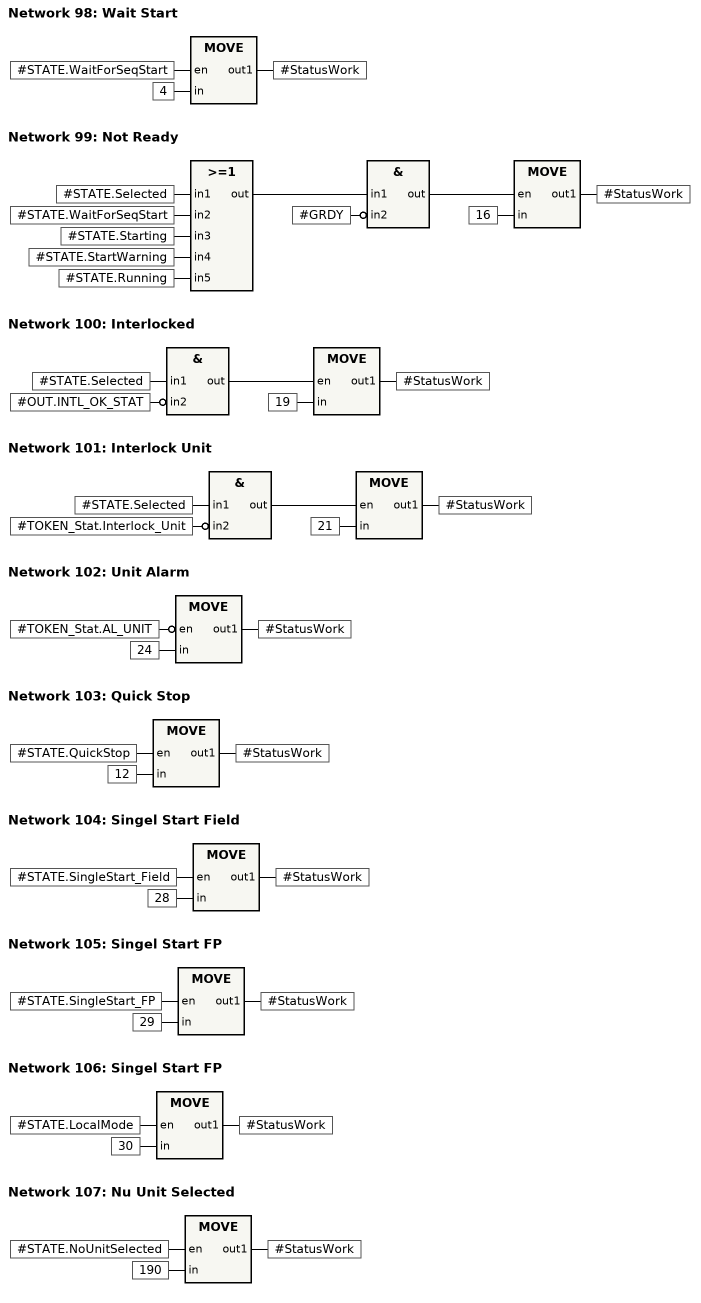
   IF #STATE.WaitForSeqStart THEN #StatusWork := 4; END_IF;
END_REGION

REGION Network 99: Not Ready
   IF (#STATE.Selected OR #STATE.WaitForSeqStart OR #STATE.Starting OR #STATE.StartWarning OR #STATE.Running) AND NOT #GRDY THEN
       #StatusWork := 16;
   END_IF;
END_REGION

REGION Network 100: Interlocked
   IF #STATE.Selected AND NOT #OUT.INTL_OK_STAT THEN #StatusWork := 19; END_IF;
END_REGION

REGION Network 101: Interlock Unit
   IF #STATE.Selected AND NOT #TOKEN_Stat.Interlock_Unit THEN #StatusWork := 21; END_IF;
END_REGION

REGION Network 102: Unit Alarm
   IF NOT #TOKEN_Stat.AL_UNIT THEN #StatusWork := 24; END_IF;
END_REGION

REGION Network 103: Quick Stop
   IF #STATE.QuickStop THEN #StatusWork := 12; END_IF;
END_REGION

REGION Network 104: Singel Start Field
   IF #STATE.SingleStart_Field THEN #StatusWork := 28; END_IF;
END_REGION

REGION Network 105: Singel Start FP
   IF #STATE.SingleStart_FP THEN #StatusWork := 29; END_IF;
END_REGION

REGION Network 106: Singel Start FP
   IF #STATE.LocalMode THEN #StatusWork := 30; END_IF;
END_REGION

REGION Network 107: Nu Unit Selected
   IF #STATE.NoUnitSelected THEN #StatusWork := 190; END_IF;
END_REGION

REGION Network 108: No CTRL Unit
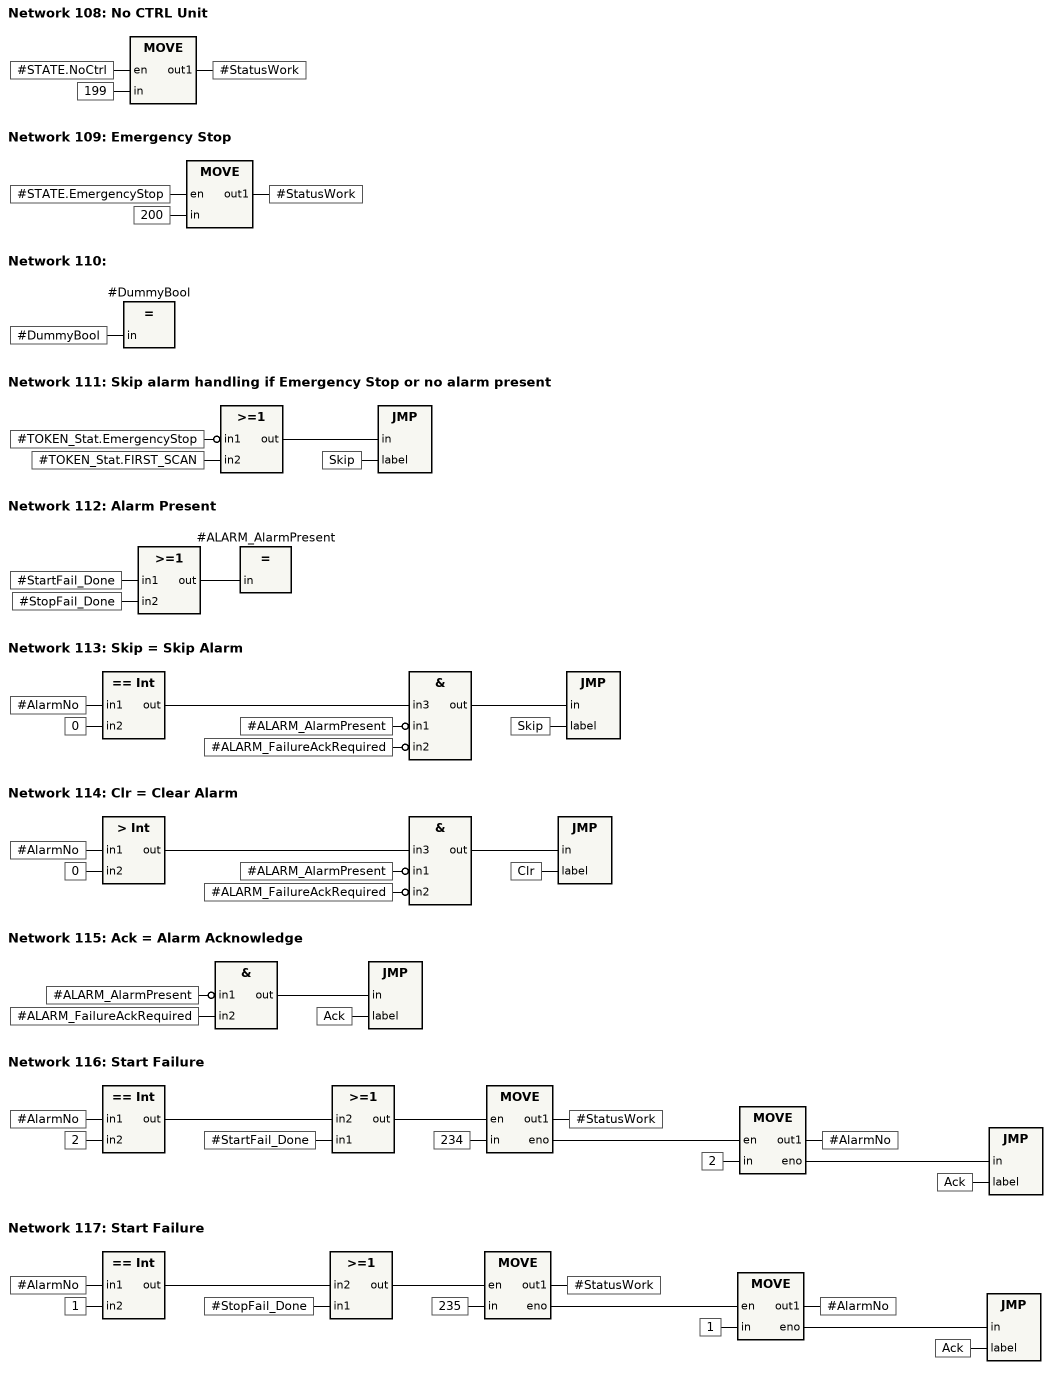
   IF #STATE.NoCtrl THEN #StatusWork := 199; END_IF;
END_REGION

REGION Network 109: Emergency Stop
   IF #STATE.EmergencyStop THEN #StatusWork := 200; END_IF;
END_REGION

REGION Network 110
   NoSt:
   #DummyBool := #DummyBool;
END_REGION

REGION Network 111: Skip alarm handling if Emergency Stop or no alarm present
   // Skip = Skip Alarm
   IF NOT #TOKEN_Stat.EmergencyStop OR #TOKEN_Stat.FIRST_SCAN THEN GOTO Skip; END_IF;
END_REGION

REGION Network 112: Alarm Present
   #ALARM_AlarmPresent := #StartFail_Done OR #StopFail_Done;
END_REGION

REGION Network 113: Skip = Skip Alarm
   IF (#AlarmNo = 0) AND NOT #ALARM_AlarmPresent AND NOT #ALARM_FailureAckRequired THEN GOTO Skip; END_IF;
END_REGION

REGION Network 114: Clr = Clear Alarm
   IF (#AlarmNo > 0) AND NOT #ALARM_AlarmPresent AND NOT #ALARM_FailureAckRequired THEN GOTO Clr; END_IF;
END_REGION

REGION Network 115: Ack = Alarm Acknowledge
   IF NOT #ALARM_AlarmPresent AND #ALARM_FailureAckRequired THEN GOTO Ack; END_IF;
END_REGION

REGION Network 116: Start Failure
   // ENO of a box is taken as its EN; it also drops when the box reports an error
   #_w1 := (#AlarmNo = 2) OR #StartFail_Done;
   IF #_w1 THEN
       #StatusWork := 234;
       #AlarmNo := 2;
       GOTO Ack;
   END_IF;
END_REGION

REGION Network 117: Start Failure
   // ENO of a box is taken as its EN; it also drops when the box reports an error
   #_w1 := (#AlarmNo = 1) OR #StopFail_Done;
   IF #_w1 THEN
       #StatusWork := 235;
       #AlarmNo := 1;
       GOTO Ack;
   END_IF;
END_REGION

REGION Network 118: Alarm Acknowledge
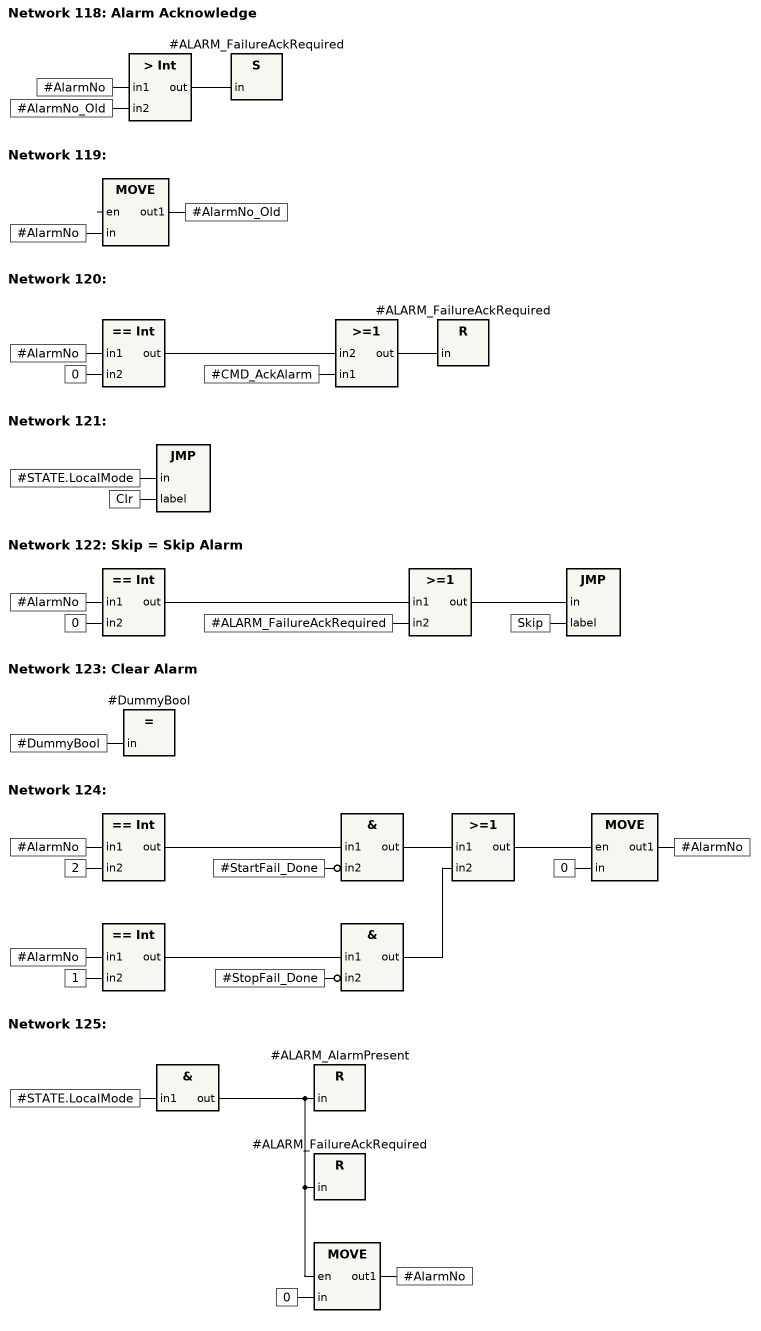
   Ack:
   IF #AlarmNo > #AlarmNo_Old THEN #ALARM_FailureAckRequired := TRUE; END_IF;
END_REGION

REGION Network 119
   #AlarmNo_Old := #AlarmNo;
END_REGION

REGION Network 120
   IF (#AlarmNo = 0) OR #CMD_AckAlarm THEN #ALARM_FailureAckRequired := FALSE; END_IF;
END_REGION

REGION Network 121
   IF #STATE.LocalMode THEN GOTO Clr; END_IF;
END_REGION

REGION Network 122: Skip = Skip Alarm
   IF (#AlarmNo = 0) OR #ALARM_FailureAckRequired THEN GOTO Skip; END_IF;
END_REGION

REGION Network 123: Clear Alarm
   Clr:
   #DummyBool := #DummyBool;
END_REGION

REGION Network 124
   IF ((#AlarmNo = 2) AND NOT #StartFail_Done) OR ((#AlarmNo = 1) AND NOT #StopFail_Done) THEN
       #AlarmNo := 0;
   END_IF;
END_REGION

REGION Network 125
   IF #STATE.LocalMode THEN
       #ALARM_AlarmPresent := FALSE;
       #ALARM_FailureAckRequired := FALSE;
       #AlarmNo := 0;
   END_IF;
END_REGION

REGION Network 126
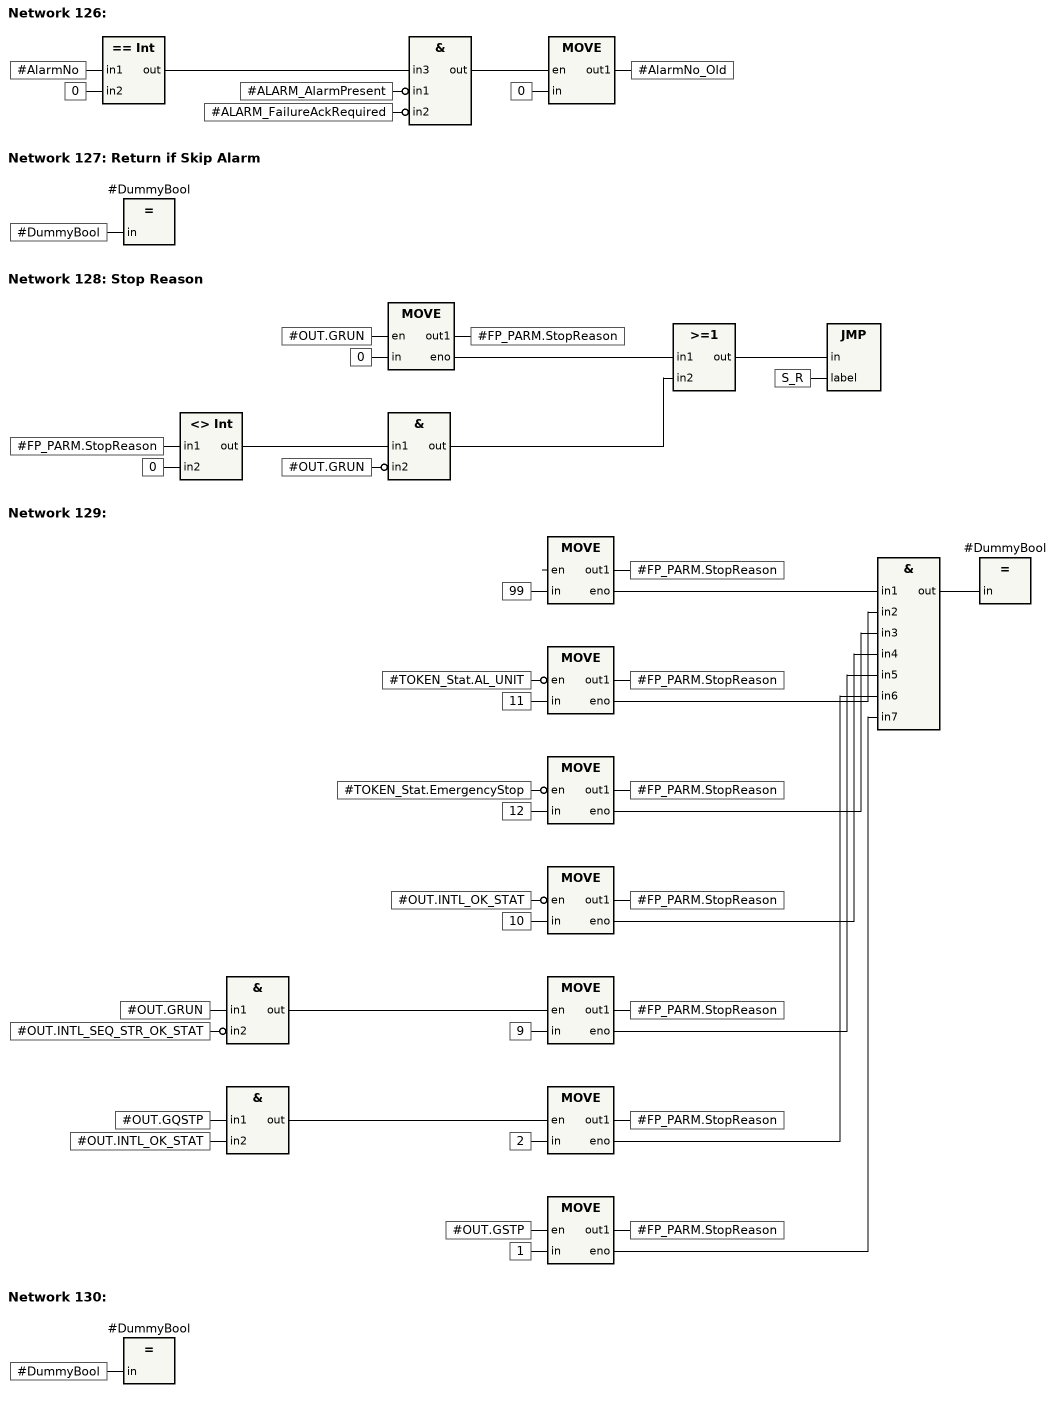
   IF (#AlarmNo = 0) AND NOT #ALARM_AlarmPresent AND NOT #ALARM_FailureAckRequired THEN
       #AlarmNo_Old := 0;
   END_IF;
END_REGION

REGION Network 127: Return if Skip Alarm
   Skip:
   #DummyBool := #DummyBool;
END_REGION

REGION Network 128: Stop Reason
   // ENO of a box is taken as its EN; it also drops when the box reports an error
   IF #OUT.GRUN THEN #FP_PARM.StopReason := 0; END_IF;
   IF #OUT.GRUN OR ((#FP_PARM.StopReason <> 0) AND NOT #OUT.GRUN) THEN GOTO S_R; END_IF;
END_REGION

REGION Network 129
   // 0 = In Operation
   // 1 = Normal Stop
   // 2 = Quick Stop
   // 10= Interlock
   // 12= Emergency Stop
   // 99= Unknown Reason
   // ENO of a box is taken as its EN; it also drops when the box reports an error
   #FP_PARM.StopReason := 99;
   IF NOT #TOKEN_Stat.AL_UNIT THEN #FP_PARM.StopReason := 11; END_IF;
   IF NOT #TOKEN_Stat.EmergencyStop THEN #FP_PARM.StopReason := 12; END_IF;
   IF NOT #OUT.INTL_OK_STAT THEN #FP_PARM.StopReason := 10; END_IF;
   #_w1 := #OUT.GRUN AND NOT #OUT.INTL_SEQ_STR_OK_STAT;
   IF #_w1 THEN #FP_PARM.StopReason := 9; END_IF;
   #_w2 := #OUT.GQSTP AND #OUT.INTL_OK_STAT;
   IF #_w2 THEN #FP_PARM.StopReason := 2; END_IF;
   IF #OUT.GSTP THEN #FP_PARM.StopReason := 1; END_IF;
   #DummyBool := NOT #TOKEN_Stat.AL_UNIT AND NOT #TOKEN_Stat.EmergencyStop AND NOT #OUT.INTL_OK_STAT AND #_w1 AND #_w2 AND #OUT.GSTP;
END_REGION

REGION Network 130
   S_R:
   #DummyBool := #DummyBool;
END_REGION

REGION Network 131: >>>> MSW to HMI <<<<<
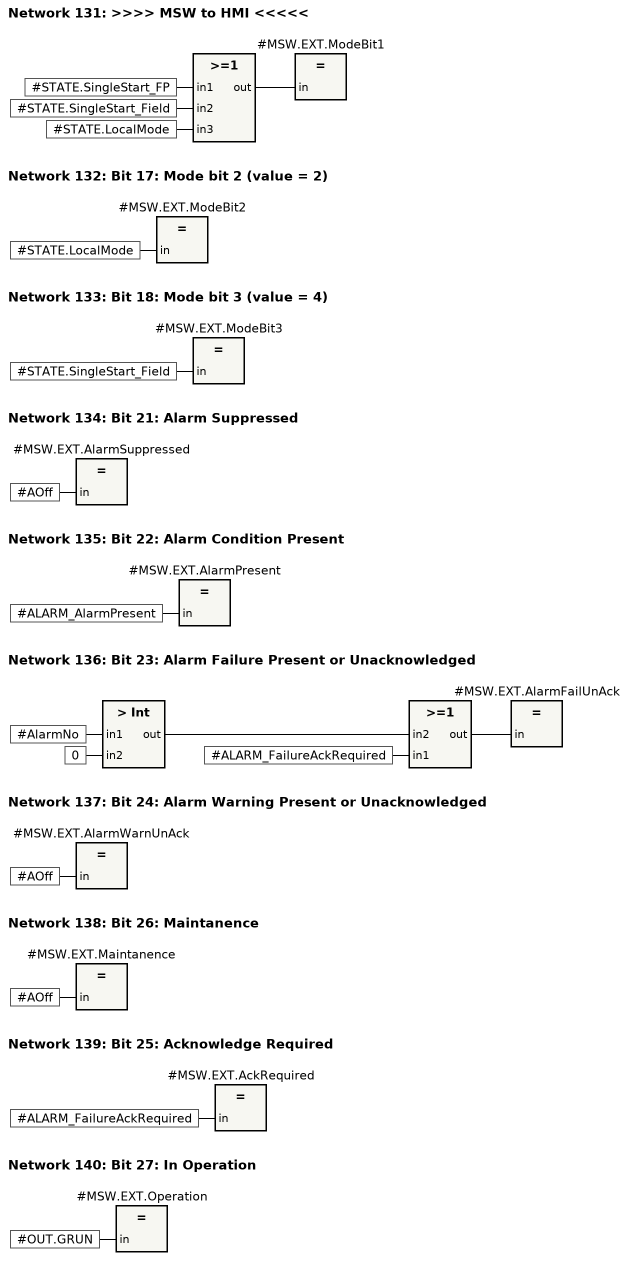
   #MSW.EXT.ModeBit1 := #STATE.SingleStart_FP OR #STATE.SingleStart_Field OR #STATE.LocalMode;
END_REGION

REGION Network 132: Bit 17: Mode bit 2 (value = 2)
   #MSW.EXT.ModeBit2 := #STATE.LocalMode;
END_REGION

REGION Network 133: Bit 18: Mode bit 3 (value = 4)
   #MSW.EXT.ModeBit3 := #STATE.SingleStart_Field;
END_REGION

REGION Network 134: Bit 21: Alarm Suppressed
   #MSW.EXT.AlarmSuppressed := #AOff;
END_REGION

REGION Network 135: Bit 22: Alarm Condition Present
   #MSW.EXT.AlarmPresent := #ALARM_AlarmPresent;
END_REGION

REGION Network 136: Bit 23: Alarm Failure Present or Unacknowledged
   #MSW.EXT.AlarmFailUnAck := (#AlarmNo > 0) OR #ALARM_FailureAckRequired;
END_REGION

REGION Network 137: Bit 24: Alarm Warning Present or Unacknowledged
   #MSW.EXT.AlarmWarnUnAck := #AOff;
END_REGION

REGION Network 138: Bit 26: Maintanence
   #MSW.EXT.Maintanence := #AOff;
END_REGION

REGION Network 139: Bit 25: Acknowledge Required
   #MSW.EXT.AckRequired := #ALARM_FailureAckRequired;
END_REGION

REGION Network 140: Bit 27: In Operation
   // Build 003 - 24.Jun.2020 (MIA-US): Replaced logic with GRUN flag
   #MSW.EXT.Operation := #OUT.GRUN;
END_REGION

REGION Network 141: Add Status to ECS status word
   // Bit 15 = 32768
   // Bit 14 = 16384
   // Bit 13 = 8192
   // Bit 12 = 4096
   // Bit 11 = 2048
   // Bit 10 = 1024
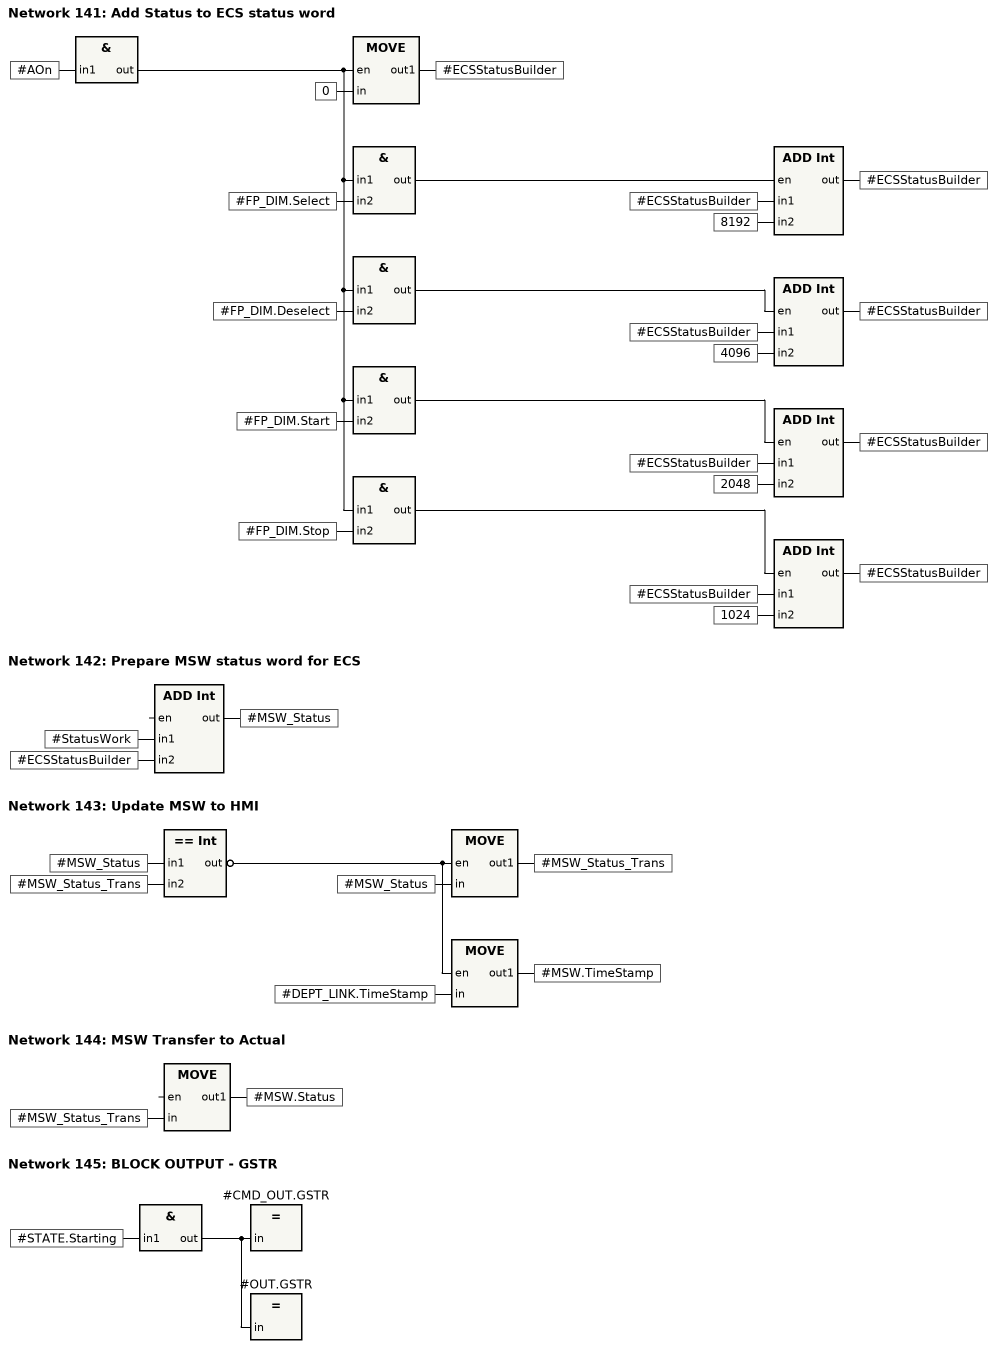
   IF #AOn THEN #ECSStatusBuilder := 0; END_IF;
   IF #AOn AND #FP_DIM.Select THEN #ECSStatusBuilder := #ECSStatusBuilder + 8192; END_IF;
   IF #AOn AND #FP_DIM.Deselect THEN #ECSStatusBuilder := #ECSStatusBuilder + 4096; END_IF;
   IF #AOn AND #FP_DIM.Start THEN #ECSStatusBuilder := #ECSStatusBuilder + 2048; END_IF;
   IF #AOn AND #FP_DIM.Stop THEN #ECSStatusBuilder := #ECSStatusBuilder + 1024; END_IF;
END_REGION

REGION Network 142: Prepare MSW status word for ECS
   #MSW_Status := #StatusWork + #ECSStatusBuilder;
END_REGION

REGION Network 143: Update MSW to HMI
   #_w1 := NOT (#MSW_Status = #MSW_Status_Trans);
   IF #_w1 THEN
       #MSW_Status_Trans := #MSW_Status;
       #MSW.TimeStamp := #DEPT_LINK.TimeStamp;
   END_IF;
END_REGION

REGION Network 144: MSW Transfer to Actual
   #MSW.Status := #MSW_Status_Trans;
END_REGION

REGION Network 145: BLOCK OUTPUT - GSTR
   #CMD_OUT.GSTR := #STATE.Starting;
   #OUT.GSTR := #STATE.Starting;
END_REGION

REGION Network 146: BLOCK OUTPUT - GSTP
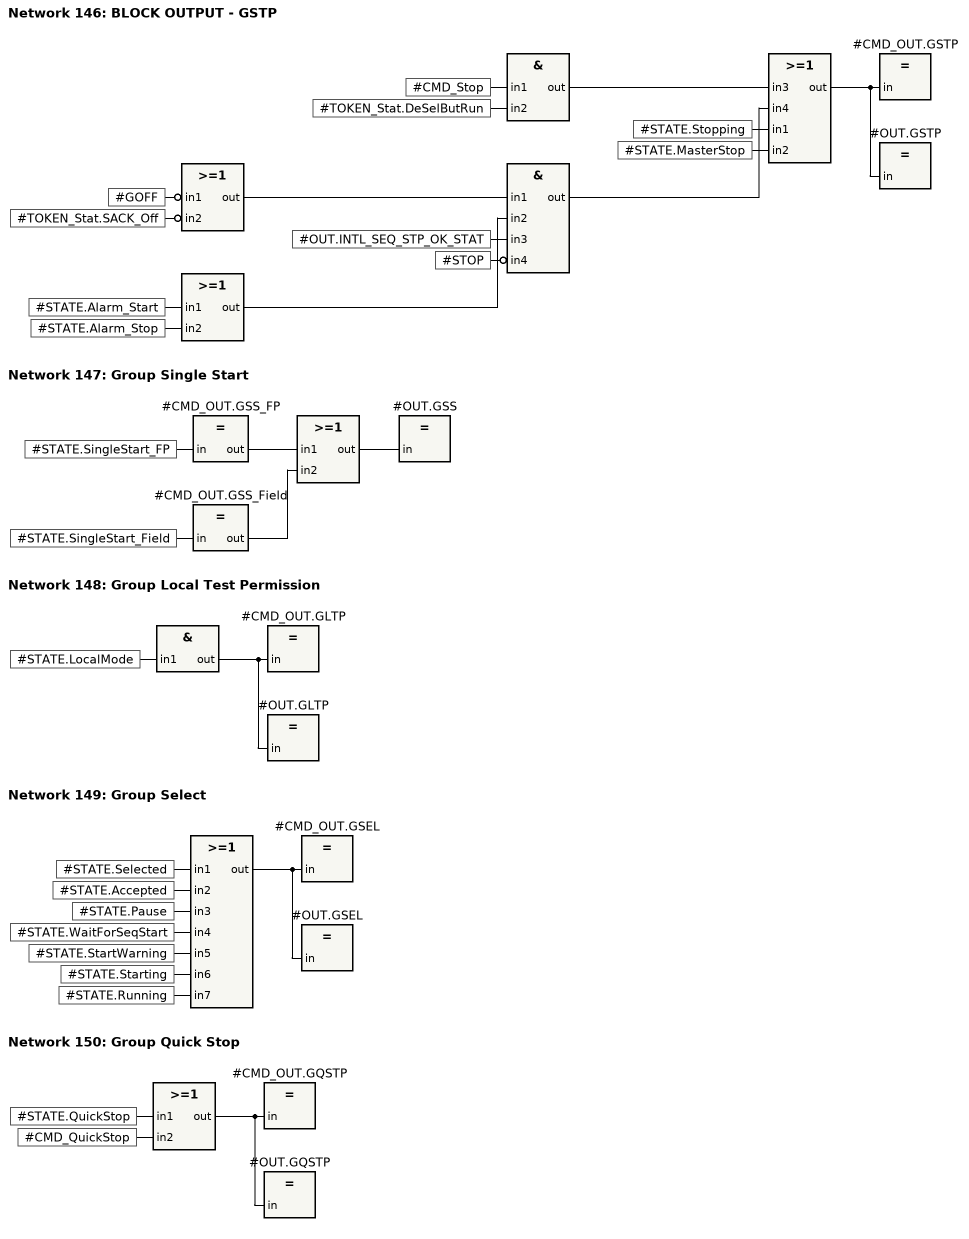
   #CMD_OUT.GSTP := (#CMD_Stop AND #TOKEN_Stat.DeSelButRun) OR ((NOT #GOFF OR NOT #TOKEN_Stat.SACK_Off) AND (#STATE.Alarm_Start OR #STATE.Alarm_Stop) AND #OUT.INTL_SEQ_STP_OK_STAT AND NOT #STOP) OR #STATE.Stopping OR #STATE.MasterStop;
   #OUT.GSTP := #CMD_OUT.GSTP;
END_REGION

REGION Network 147: Group Single Start
   #CMD_OUT.GSS_FP := #STATE.SingleStart_FP;
   #CMD_OUT.GSS_Field := #STATE.SingleStart_Field;
   #OUT.GSS := #STATE.SingleStart_FP OR #STATE.SingleStart_Field;
END_REGION

REGION Network 148: Group Local Test Permission
   #CMD_OUT.GLTP := #STATE.LocalMode;
   #OUT.GLTP := #STATE.LocalMode;
END_REGION

REGION Network 149: Group Select
   #CMD_OUT.GSEL := #STATE.Selected OR #STATE.Accepted OR #STATE.Pause OR #STATE.WaitForSeqStart OR #STATE.StartWarning OR #STATE.Starting OR #STATE.Running;
   #OUT.GSEL := #CMD_OUT.GSEL;
END_REGION

REGION Network 150: Group Quick Stop
   #CMD_OUT.GQSTP := #STATE.QuickStop OR #CMD_QuickStop;
   #OUT.GQSTP := #CMD_OUT.GQSTP;
END_REGION

REGION Network 151: Accepted
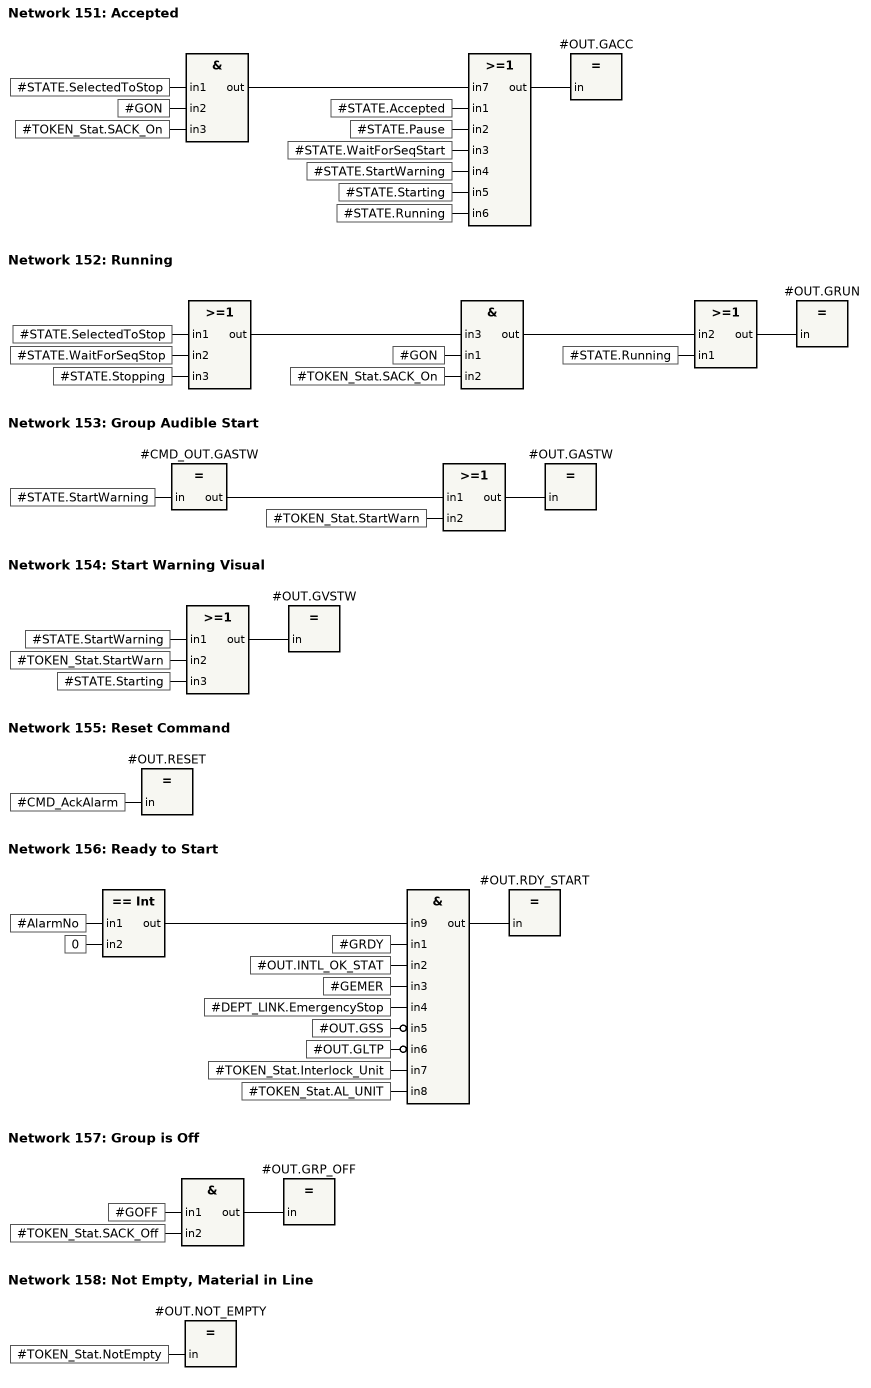
   #OUT.GACC := (#STATE.SelectedToStop AND #GON AND #TOKEN_Stat.SACK_On) OR #STATE.Accepted OR #STATE.Pause OR #STATE.WaitForSeqStart OR #STATE.StartWarning OR #STATE.Starting OR #STATE.Running;
END_REGION

REGION Network 152: Running
   // Build 003 - 24.Jun.2020 (MIA-US): Reworked logic
   #OUT.GRUN := ((#STATE.SelectedToStop OR #STATE.WaitForSeqStop OR #STATE.Stopping) AND #GON AND #TOKEN_Stat.SACK_On) OR #STATE.Running;
END_REGION

REGION Network 153: Group Audible Start
   #CMD_OUT.GASTW := #STATE.StartWarning;
   #OUT.GASTW := #STATE.StartWarning OR #TOKEN_Stat.StartWarn;
END_REGION

REGION Network 154: Start Warning Visual
   #OUT.GVSTW := #STATE.StartWarning OR #TOKEN_Stat.StartWarn OR #STATE.Starting;
END_REGION

REGION Network 155: Reset Command
   #OUT.RESET := #CMD_AckAlarm;
END_REGION

REGION Network 156: Ready to Start
   #OUT.RDY_START := (#AlarmNo = 0) AND #GRDY AND #OUT.INTL_OK_STAT AND #GEMER AND #DEPT_LINK.EmergencyStop AND NOT #OUT.GSS AND NOT #OUT.GLTP AND #TOKEN_Stat.Interlock_Unit AND #TOKEN_Stat.AL_UNIT;
END_REGION

REGION Network 157: Group is Off
   #OUT.GRP_OFF := #GOFF AND #TOKEN_Stat.SACK_Off;
END_REGION

REGION Network 158: Not Empty, Material in Line
   #OUT.NOT_EMPTY := #TOKEN_Stat.NotEmpty;
END_REGION

REGION Network 159: PASS INFO BACK TO DEPARTMENT - All Group On
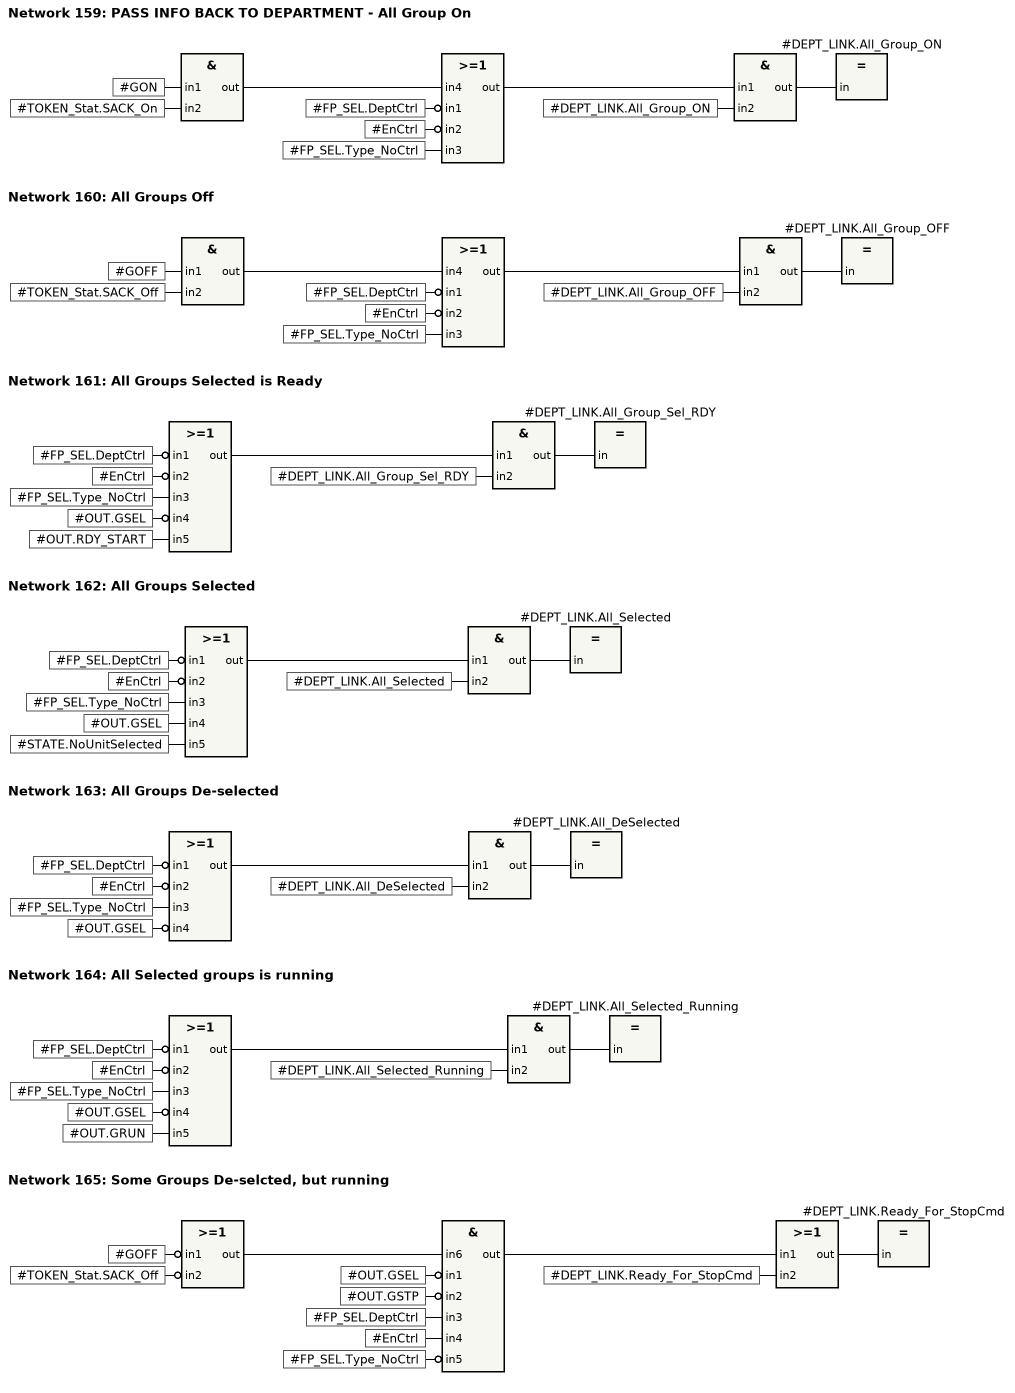
   #DEPT_LINK.All_Group_ON := ((#GON AND #TOKEN_Stat.SACK_On) OR NOT #FP_SEL.DeptCtrl OR NOT #EnCtrl OR #FP_SEL.Type_NoCtrl) AND #DEPT_LINK.All_Group_ON;
END_REGION

REGION Network 160: All Groups Off
   #DEPT_LINK.All_Group_OFF := ((#GOFF AND #TOKEN_Stat.SACK_Off) OR NOT #FP_SEL.DeptCtrl OR NOT #EnCtrl OR #FP_SEL.Type_NoCtrl) AND #DEPT_LINK.All_Group_OFF;
END_REGION

REGION Network 161: All Groups Selected is Ready
   #DEPT_LINK.All_Group_Sel_RDY := (NOT #FP_SEL.DeptCtrl OR NOT #EnCtrl OR #FP_SEL.Type_NoCtrl OR NOT #OUT.GSEL OR #OUT.RDY_START) AND #DEPT_LINK.All_Group_Sel_RDY;
END_REGION

REGION Network 162: All Groups Selected
   #DEPT_LINK.All_Selected := (NOT #FP_SEL.DeptCtrl OR NOT #EnCtrl OR #FP_SEL.Type_NoCtrl OR #OUT.GSEL OR #STATE.NoUnitSelected) AND #DEPT_LINK.All_Selected;
END_REGION

REGION Network 163: All Groups De-selected
   #DEPT_LINK.All_DeSelected := (NOT #FP_SEL.DeptCtrl OR NOT #EnCtrl OR #FP_SEL.Type_NoCtrl OR NOT #OUT.GSEL) AND #DEPT_LINK.All_DeSelected;
END_REGION

REGION Network 164: All Selected groups is running
   #DEPT_LINK.All_Selected_Running := (NOT #FP_SEL.DeptCtrl OR NOT #EnCtrl OR #FP_SEL.Type_NoCtrl OR NOT #OUT.GSEL OR #OUT.GRUN) AND #DEPT_LINK.All_Selected_Running;
END_REGION

REGION Network 165: Some Groups De-selcted, but running
   #DEPT_LINK.Ready_For_StopCmd := ((NOT #GOFF OR NOT #TOKEN_Stat.SACK_Off) AND NOT #OUT.GSEL AND NOT #OUT.GSTP AND #FP_SEL.DeptCtrl AND #EnCtrl AND NOT #FP_SEL.Type_NoCtrl) OR #DEPT_LINK.Ready_For_StopCmd;
END_REGION

REGION Network 166: TOKEN PASSING
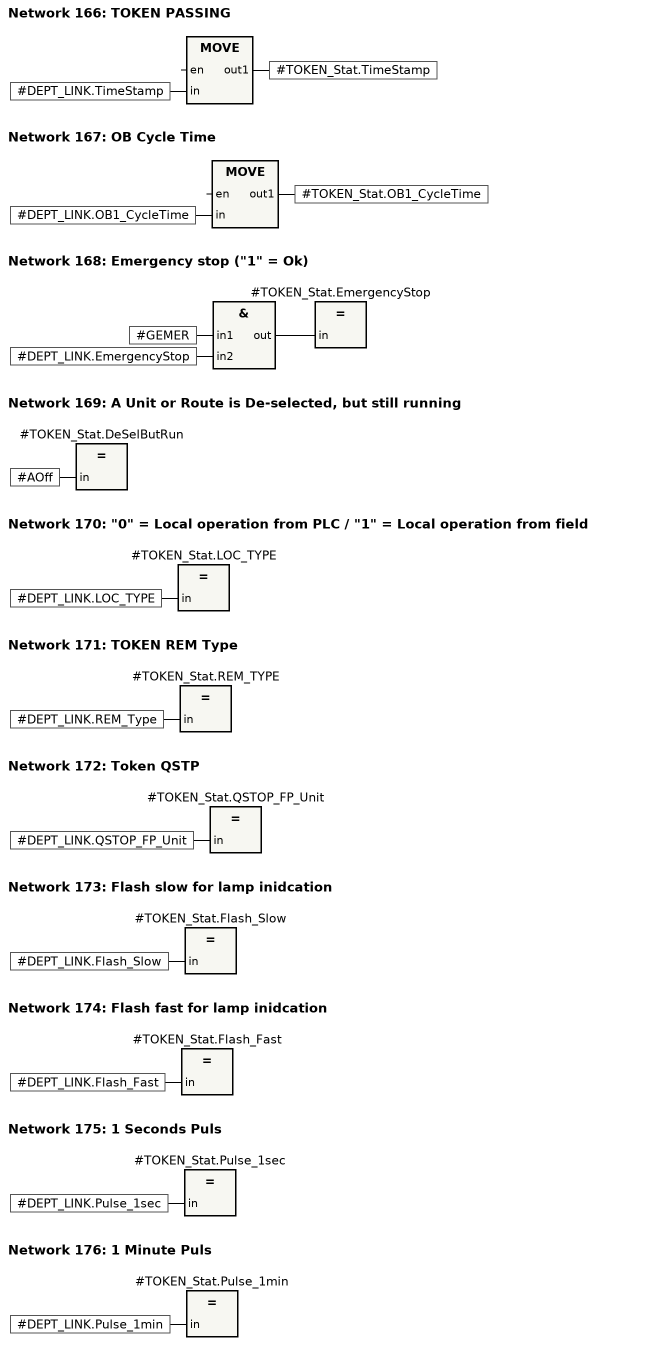
   #TOKEN_Stat.TimeStamp := #DEPT_LINK.TimeStamp;
END_REGION

REGION Network 167: OB Cycle Time
   #TOKEN_Stat.OB1_CycleTime := #DEPT_LINK.OB1_CycleTime;
END_REGION

REGION Network 168: Emergency stop ("1" = Ok)
   #TOKEN_Stat.EmergencyStop := #GEMER AND #DEPT_LINK.EmergencyStop;
END_REGION

REGION Network 169: A Unit or Route is De-selected, but still running
   #TOKEN_Stat.DeSelButRun := #AOff;
END_REGION

REGION Network 170: "0" = Local operation from PLC / "1" = Local operation from field
   #TOKEN_Stat.LOC_TYPE := #DEPT_LINK.LOC_TYPE;
END_REGION

REGION Network 171: TOKEN REM Type
   #TOKEN_Stat.REM_TYPE := #DEPT_LINK.REM_Type;
END_REGION

REGION Network 172: Token QSTP
   #TOKEN_Stat.QSTOP_FP_Unit := #DEPT_LINK.QSTOP_FP_Unit;
END_REGION

REGION Network 173: Flash slow for lamp inidcation
   #TOKEN_Stat.Flash_Slow := #DEPT_LINK.Flash_Slow;
END_REGION

REGION Network 174: Flash fast for lamp inidcation
   #TOKEN_Stat.Flash_Fast := #DEPT_LINK.Flash_Fast;
END_REGION

REGION Network 175: 1 Seconds Puls
   #TOKEN_Stat.Pulse_1sec := #DEPT_LINK.Pulse_1sec;
END_REGION

REGION Network 176: 1 Minute Puls
   #TOKEN_Stat.Pulse_1min := #DEPT_LINK.Pulse_1min;
END_REGION

REGION Network 177: 1 Hour Puls
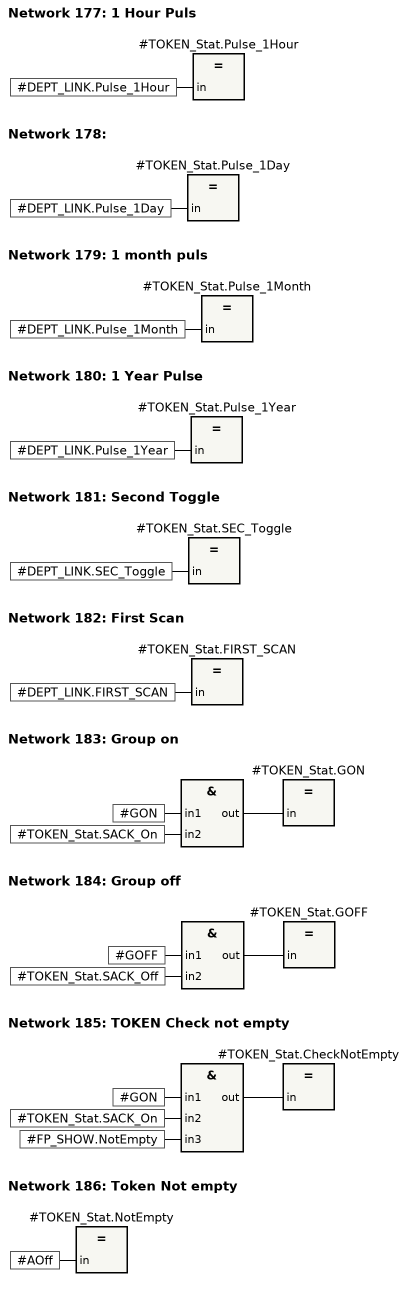
   #TOKEN_Stat.Pulse_1Hour := #DEPT_LINK.Pulse_1Hour;
END_REGION

REGION Network 178
   #TOKEN_Stat.Pulse_1Day := #DEPT_LINK.Pulse_1Day;
END_REGION

REGION Network 179: 1 month puls
   #TOKEN_Stat.Pulse_1Month := #DEPT_LINK.Pulse_1Month;
END_REGION

REGION Network 180: 1 Year Pulse
   #TOKEN_Stat.Pulse_1Year := #DEPT_LINK.Pulse_1Year;
END_REGION

REGION Network 181: Second Toggle
   #TOKEN_Stat.SEC_Toggle := #DEPT_LINK.SEC_Toggle;
END_REGION

REGION Network 182: First Scan
   #TOKEN_Stat.FIRST_SCAN := #DEPT_LINK.FIRST_SCAN;
END_REGION

REGION Network 183: Group on
   #TOKEN_Stat.GON := #GON AND #TOKEN_Stat.SACK_On;
END_REGION

REGION Network 184: Group off
   #TOKEN_Stat.GOFF := #GOFF AND #TOKEN_Stat.SACK_Off;
END_REGION

REGION Network 185: TOKEN Check not empty
   #TOKEN_Stat.CheckNotEmpty := #GON AND #TOKEN_Stat.SACK_On AND #FP_SHOW.NotEmpty;
END_REGION

REGION Network 186: Token Not empty
   #TOKEN_Stat.NotEmpty := #AOff;
END_REGION

REGION Network 187: TOKEN Reset not empty
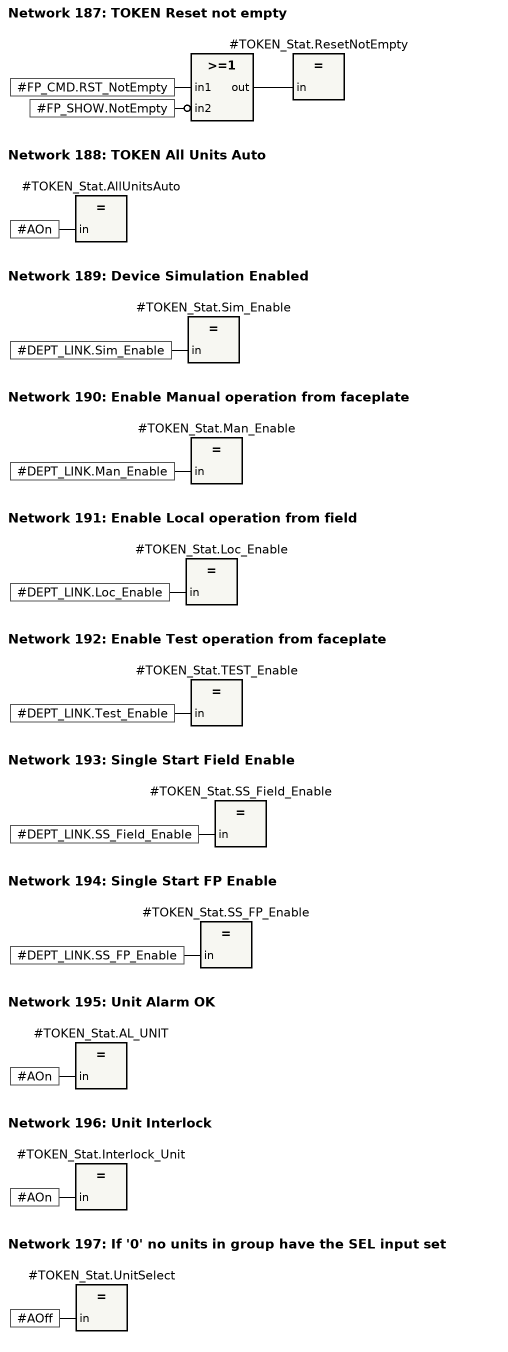
   #TOKEN_Stat.ResetNotEmpty := #FP_CMD.RST_NotEmpty OR NOT #FP_SHOW.NotEmpty;
END_REGION

REGION Network 188: TOKEN All Units Auto
   #TOKEN_Stat.AllUnitsAuto := #AOn;
END_REGION

REGION Network 189: Device Simulation Enabled
   #TOKEN_Stat.Sim_Enable := #DEPT_LINK.Sim_Enable;
END_REGION

REGION Network 190: Enable Manual operation from faceplate
   #TOKEN_Stat.Man_Enable := #DEPT_LINK.Man_Enable;
END_REGION

REGION Network 191: Enable Local operation from field
   #TOKEN_Stat.Loc_Enable := #DEPT_LINK.Loc_Enable;
END_REGION

REGION Network 192: Enable Test operation from faceplate
   #TOKEN_Stat.TEST_Enable := #DEPT_LINK.Test_Enable;
END_REGION

REGION Network 193: Single Start Field Enable
   #TOKEN_Stat.SS_Field_Enable := #DEPT_LINK.SS_Field_Enable;
END_REGION

REGION Network 194: Single Start FP Enable
   #TOKEN_Stat.SS_FP_Enable := #DEPT_LINK.SS_FP_Enable;
END_REGION

REGION Network 195: Unit Alarm OK
   #TOKEN_Stat.AL_UNIT := #AOn;
END_REGION

REGION Network 196: Unit Interlock
   #TOKEN_Stat.Interlock_Unit := #AOn;
END_REGION

REGION Network 197: If '0' no units in group have the SEL input set
   #TOKEN_Stat.UnitSelect := #AOff;
END_REGION

REGION Network 198: Alarm Suppression
